Universal Robots URScript: samho_main_Fillet_2023_10_18.script

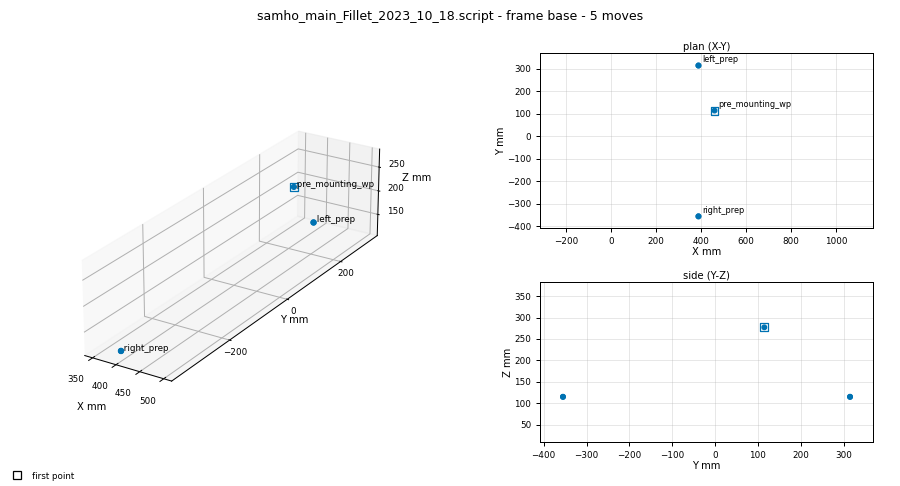
[picture p0: tool path of samho_main_Fillet_2023_10_18.script in frame base, 5 of 121 moves have a stored position in this frame; points joined in program order, loops and branches not executed]
def samho_main_Fillet_2023_10_18():
  set_gravity([0.0, 0.0, 9.82])
  set_standard_analog_input_domain(0, 1)
  set_standard_analog_input_domain(1, 1)
  set_tool_analog_input_domain(0, 1)
  set_tool_analog_input_domain(1, 1)
  set_analog_outputdomain(0, 1)
  set_analog_outputdomain(1, 1)
  set_input_actions_to_default()
  set_tool_digital_input_action(1, "freedrive")
  set_runstate_standard_digital_outputs([0])
  set_runstate_standard_digital_output_to_value(0, 1)
  set_runstate_standard_digital_output_to_value(7, 3)
  step_count_c3da284d_8c38_4948_9d0a_7bbcd1285130 = 0.0
  thread Step_Counter_Thread_b1fbcd7f_a7e8_4366_aae2_1cd96c806efd():
    while (True):
      step_count_c3da284d_8c38_4948_9d0a_7bbcd1285130 = step_count_c3da284d_8c38_4948_9d0a_7bbcd1285130 + 1.0
      sync()
    end
  end
  run Step_Counter_Thread_b1fbcd7f_a7e8_4366_aae2_1cd96c806efd()
  set_safety_mode_transition_hardness(1)
  set_tool_voltage(24)
  set_tcp(p[-0.20748,-9.0E-4,0.38521,1.2569,0.0099,-2.8767])
  set_payload(2.4, [-0.085, 0.00191, 0.125])
  modbus_add_signal("127.0.0.1", 255, 171, 2, "MODBUS_1", False)
  modbus_set_signal_update_frequency("MODBUS_1", 1)
  modbus_add_signal("127.0.0.1", 255, 153, 2, "MODBUS_2", False)
  modbus_set_signal_update_frequency("MODBUS_2", 10)
  modbus_add_signal("127.0.0.1", 255, 154, 2, "MODBUS_3", False)
  modbus_set_signal_update_frequency("MODBUS_3", 10)
  modbus_add_signal("127.0.0.1", 255, 240, 2, "MODBUS_4", False)
  modbus_set_signal_update_frequency("MODBUS_4", 10)
  global A_Touch_trig_l=[False, False, False, False, True, False, False, False, False, False, False]
  global Auto_cur_cell=0
  global last_wv_line=p[0, 0, 0, 0, 0, 0]
  global Auto_trig=False
  global A_Touch_p=[p[0, 0, 0, 0, 0, 0], p[0, 0, 0, 0, 0, 0], p[0, 0, 0, 0, 0, 0], p[0, 0, 0, 0, 0, 0], p[0.52449, -0.29611, -0.03135, -1.44433, -1.03764, -1.44433], p[0, 0, 0, 0, 0, 0], p[0, 0, 0, 0, 0, 0], p[0, 0, 0, 0, 0, 0], p[0, 0, 0, 0, 0, 0], p[0, 0, 0, 0, 0, 0], p[0, 0, 0, 0, 0, 0], p[0, 0, 0, 0, 0, 0], p[0, 0, 0, 0, 0, 0], p[0.5215, -0.2959, 0.14321, -1.44433, -1.03764, -1.44433], p[0, 0, 0, 0, 0, 0], p[0, 0, 0, 0, 0, 0]]
  global last_wv_wp1=p[0, 0, 0, 0, 0, 0]
  global last_pose=p[0, 0, 0, 0, 0, 0]
  global A_Distance_list=[0, 0, 0, 0, 0, 0, 0, 0, 0, 0, 0, 0, 0, 0, 0, 0]
  global Auto_total_cell=1
  global Reset_Trig=False
  global A_Prepos_l=[p[0, 0, 0, 0, 0, 0], p[0, 0, 0, 0, 0, 0], p[0, 0, 0, 0, 0, 0], p[0, 0, 0, 0, 0, 0], p[0.47946, -0.33036, 0.01979, 1.89026, -1.12958, 1.54553], p[0, 0, 0, 0, 0, 0], p[0, 0, 0, 0, 0, 0], p[0, 0, 0, 0, 0, 0], p[0, 0, 0, 0, 0, 0], p[0, 0, 0, 0, 0, 0], p[0, 0, 0, 0, 0, 0], p[0, 0, 0, 0, 0, 0], p[0, 0, 0, 0, 0, 0], p[0, 0, 0, 0, 0, 0], p[0, 0, 0, 0, 0, 0], p[0, 0, 0, 0, 0, 0]]
  global last_z_bottom=0
  global A_Speed_list=[0, 0, 0, 0, 0, 0, 0, 0, 0, 0, 0, 0, 0, 0, 0, 0]
  global Auto_W_num=[4, 0, 0, 0, 0, 0, 0, 0, 0, 0, 0, 0, 0, 0, 0]
  global last_tilt_deg=[0, 0, 0]
  global Base=p[0.0,0.0,0.0,0.0,0.0,0.0]
  global save_timer=0
  global timer_1=0
  def calculate_point_to_move_towards(feature, direction, position_distance):
    local posDir=[direction[0], direction[1], direction[2]]
    if (norm(posDir) < 1e-6):
      return get_target_waypoint()
    end
    local direction_vector_normalized=normalize(posDir)
    local displacement_pose=p[direction_vector_normalized[0] * position_distance,direction_vector_normalized[1] * position_distance,direction_vector_normalized[2] * position_distance,0,0,0]
    local wanted_displacement_in_base_frame=pose_sub(pose_trans(feature, displacement_pose), feature)
    return pose_add(get_target_waypoint(), wanted_displacement_in_base_frame)
  end
  global save_timer_is_counting=False
  global timer_1_is_counting=False
  thread Timer_Thread():
    while (True):
      if (save_timer_is_counting):
        save_timer = save_timer + get_steptime()
      end
      if (timer_1_is_counting):
        timer_1 = timer_1 + get_steptime()
      end
      sync()
    end
  end
  run Timer_Thread()
  def cell_info():
    $ 1483 "cell_info" "noBreak"
    $ 1484 "'cell_setting'"
    # 'cell_setting'
    $ 1485 "a7_f_distance≔get_center"
    global a7_f_distance=get_center
    $ 1486 "'dis + 125'"
    # 'dis + 125'
    $ 1487 "If simulation_mode"
    if (simulation_mode):
      $ 1488 "a6_f_height_l≔190"
      global a6_f_height_l=190
      $ 1489 "a6_f_height_r≔190"
      global a6_f_height_r=190
      $ 1490 "a6_f_width≔690"
      global a6_f_width=690
      $ 1491 "a6_callar_hor≔100"
      global a6_callar_hor=100
      $ 1492 "a6_callar_vert≔100"
      global a6_callar_vert=100
      $ 1493 "center_height≔50"
      global center_height=50
      $ 1494 "EXT_flag1≔integer_to_binary_list(2048)"
      global EXT_flag1= integer_to_binary_list (2048)
      $ 1495 "get_margin_z≔50"
      global get_margin_z=50
    else:
      $ 1496 "Else" "noBreak"
      $ 1497 "a6_f_height_l≔read_port_register(173)"
      global a6_f_height_l= read_port_register (173)
      $ 1498 "a6_f_height_r≔read_port_register(174)"
      global a6_f_height_r= read_port_register (174)
      $ 1499 "a6_f_width≔read_port_register(175)"
      global a6_f_width= read_port_register (175)
      $ 1500 "a6_callar_hor≔read_port_register(181)"
      global a6_callar_hor= read_port_register (181)
      $ 1501 "a6_callar_vert≔read_port_register(182)"
      global a6_callar_vert= read_port_register (182)
      $ 1502 "center_height≔read_port_register(237)"
      global center_height=read_port_register(237)
      $ 1503 "EXT_flag1≔integer_to_binary_list(read_port_register(179))"
      global EXT_flag1= integer_to_binary_list ( read_port_register (179))
      $ 1505 "get_margin_z≔read_port_register(238)"
      global get_margin_z=read_port_register(238)
      $ 1507 "If center_height>32765"
      if (center_height>32765):
        $ 1508 "center_height≔center_height-65535"
        global center_height=center_height-65535
      end
      $ 1509 "If get_margin_z>32765"
      if (get_margin_z>32765):
        $ 1510 "get_margin_z≔get_margin_z-65535"
        global get_margin_z=get_margin_z-65535
      end
    end
    $ 1511 "Initialization"
    $ 1512 "CELL_ROBOT_DIST≔a7_f_distance"
    global CELL_ROBOT_DIST=a7_f_distance
    $ 1513 "CELL_WIDTH≔a6_f_width"
    global CELL_WIDTH=a6_f_width
  end
  def robotand_cell_initalizat():
    $ 1514 "robotand_cell_initalizat" "noBreak"
    $ 1515 "If Auto_trig≟ True "
    if (Auto_trig ==   True  ):
      $ 1516 "Auto_trig≔ False "
      global Auto_trig=  False
      $ 1517 "init"
      $ 1518 "write_port_register(cell_3f_2f_151,0)"
      write_port_register(cell_3f_2f_151,0)
      $ 1519 "write_port_register(cell_info_152,0)"
      write_port_register(cell_info_152,0)
      $ 1520 "write_port_register(weld_req_153,0)"
      write_port_register(weld_req_153,0)
      $ 1521 "write_port_register(touch_cell_155,0)"
      write_port_register(touch_cell_155,0)
      $ 1522 "write_port_register(touch_num_156,0)"
      write_port_register(touch_num_156,0)
      $ 1523 "write_port_register(touch_done_157,0)"
      write_port_register(touch_done_157,0)
      $ 1524 "write_port_register(weld_done_137,0)"
      write_port_register(weld_done_137,0)
      $ 1525 "write_port_register(135,0)"
      write_port_register(135,0)
      $ 1526 "write_port_register(136,0)"
      write_port_register(136,0)
      $ 1527 "write_port_register(165,0)"
      write_port_register(165,0)
      $ 1528 "write_port_register(166,0)"
      write_port_register(166,0)
      $ 1529 "write_port_register(167,0)"
      write_port_register(167,0)
      $ 1530 "write_port_register(169,0)"
      write_port_register(169,0)
      $ 1531 "write_port_register(170,0)"
      write_port_register(170,0)
      $ 1532 "write_port_register(221,0)"
      write_port_register(221,0)
      $ 1533 "write_port_register(222,0)"
      write_port_register(222,0)
      $ 1534 "write_port_register(223,0)"
      write_port_register(223,0)
      $ 1535 "write_port_register(224,0)"
      write_port_register(224,0)
      $ 1536 "write_port_register(225,0)"
      write_port_register(225,0)
      $ 1537 "write_port_register(226,0)"
      write_port_register(226,0)
      $ 1538 "write_port_register(227,0)"
      write_port_register(227,0)
      $ 1539 "write_port_register(228,0)"
      write_port_register(228,0)
      $ 1540 "write_port_register(240,0)"
      write_port_register(240,0)
      $ 1541 "write_port_register(176,0)"
      write_port_register(176,0)
      $ 1542 "write_port_register(177,0)"
      write_port_register(177,0)
      $ 1543 "write_port_register(154,0)"
      write_port_register(154,0)
    end
    $ 1544 "sync()"
    sync()
  end
  def welding_parameter_init():
    $ 1545 "welding_parameter_init" "noBreak"
    $ 1546 "init"
    $ 1547 "If A_sel_v≟A_VL1 or A_sel_v≟A_VL2 or A_sel_v≟A_VR1 or A_sel_v≟A_VR2"
    if (A_sel_v == A_VL1  or  A_sel_v == A_VL2  or  A_sel_v == A_VR1  or  A_sel_v == A_VR2):
      $ 1548 "position_3f2f≔position_3F"
      global position_3f2f=position_3F
      $ 1549 "write_port_register(cell_3f_2f_151,A_sel_v)"
      write_port_register(cell_3f_2f_151,A_sel_v)
      $ 1550 "b8_wv_2f≔ False "
      global b8_wv_2f=  False
      $ 1551 "d_lean_degree≔0"
      global d_lean_degree=0
    else:
      $ 1552 "Else" "noBreak"
      $ 1553 "position_3f2f≔position_2F"
      global position_3f2f=position_2F
      $ 1554 "b8_wv_2f≔ True "
      global b8_wv_2f=  True
      $ 1555 "d_lean_degree≔30"
      global d_lean_degree=30
      $ 1556 "write_port_register(cell_3f_2f_151,A_HOR)"
      write_port_register(cell_3f_2f_151,A_HOR)
    end
    $ 1557 "If current_path≥2"
    if (current_path >= 2):
      $ 1558 "write_port_register(cell_info_152,current_path)"
      write_port_register(cell_info_152,current_path)
    else:
      $ 1559 "Else" "noBreak"
      $ 1560 "write_port_register(cell_info_152,1)"
      write_port_register(cell_info_152,1)
    end
    $ 1561 "write_port_register(return_done_240,0)"
    write_port_register(return_done_240,0)
    $ 1562 "Wait: 0.3"
    sleep(0.3)
    $ 1563 "write_port_register(weld_req_153,1)"
    write_port_register(weld_req_153,1)
    $ 1564 "Wait read_port_register(return_done_240)≟1"
    while (not( read_port_register (return_done_240) == 1)):
      sync()
    end
    $ 1565 "write_port_register(weld_req_153,0)"
    write_port_register(weld_req_153,0)
    $ 1566 "touch_m_check≔0"
    global touch_m_check=0
    $ 1567 "start_end_from_pendant"
    $ 1568 "d_start_current≔read_port_register(244)/10"
    global d_start_current= read_port_register (244)/10
    $ 1569 "d_start_voltage≔read_port_register(245)/10"
    global d_start_voltage= read_port_register (245)/10
    $ 1570 "d_start_time≔read_port_register(241)/10"
    global d_start_time= read_port_register (241)/10
    $ 1571 "d_end_current≔read_port_register(249)/10"
    global d_end_current= read_port_register (249)/10
    $ 1572 "d_end_voltage≔read_port_register(250)/10"
    global d_end_voltage= read_port_register (250)/10
    $ 1573 "d_end_time≔read_port_register(246)/10"
    global d_end_time= read_port_register (246)/10
    $ 1574 "d_end_current_2≔read_port_register(254)/10"
    global d_end_current_2= read_port_register (254)/10
    $ 1575 "d_end_voltage_2≔read_port_register(255)/10"
    global d_end_voltage_2= read_port_register (255)/10
    $ 1576 "d_end_time_2≔read_port_register(251)/10"
    global d_end_time_2= read_port_register (251)/10
    $ 1577 "a7_weld_crater≔[d_start_current,d_start_voltage,d_start_time,d_end_current,d_end_voltage,d_end_time,d_lean_degree]"
    global a7_weld_crater=[d_start_current,d_start_voltage,d_start_time,d_end_current,d_end_voltage,d_end_time,d_lean_degree]
    $ 1578 "a0_volt_ref≔read_port_register(231)/10"
    global a0_volt_ref= read_port_register (231)/10
    $ 1579 "a1_amp_ref≔read_port_register(232)/10"
    global a1_amp_ref= read_port_register (232)/10
    $ 1580 "a2_speed_cpm≔read_port_register(233)/10"
    global a2_speed_cpm= read_port_register (233)/10
    $ 1581 "a3_wv_amplitude≔read_port_register(234)/10"
    global a3_wv_amplitude= read_port_register (234)/10
    $ 1582 "a4_wv_frequency≔read_port_register(225)/10"
    global a4_wv_frequency= read_port_register (225)/10
    $ 1583 "b1_appro_param≔0"
    global b1_appro_param=0
    $ 1584 "b4_wv_delay2≔read_port_register(226)/10"
    global b4_wv_delay2= read_port_register (226)/10
    $ 1585 "b6_wv_delay4≔read_port_register(227)/10"
    global b6_wv_delay4= read_port_register (227)/10
    $ 1586 "b3_wv_delay1≔0"
    global b3_wv_delay1=0
    $ 1587 "b5_wv_delay3≔0"
    global b5_wv_delay3=0
    $ 1588 "b3_dealy_all≔[b3_wv_delay1,b4_wv_delay2,b5_wv_delay3,b6_wv_delay4]"
    global b3_dealy_all=[b3_wv_delay1,b4_wv_delay2,b5_wv_delay3,b6_wv_delay4]
    $ 1589 "get_width_182≔read_port_register(182)"
    global get_width_182= read_port_register (182)
    $ 1590 "b9_touch_sens≔20"
    global b9_touch_sens=20
    $ 1591 "task_angle≔register_read(228)/10"
    global task_angle=register_read(228)/10
    $ 1592 "Circle_Speed≔a2_speed_cpm"
    global Circle_Speed=a2_speed_cpm
    $ 1593 "CELL_BOTTOM≔a7_cell_bottom"
    global CELL_BOTTOM=a7_cell_bottom
    $ 1594 "a6_scallup_left≔read_port_register(176)"
    global a6_scallup_left= read_port_register (176)
    $ 1595 "a6_scallup_righ≔read_port_register(177)"
    global a6_scallup_righ= read_port_register (177)
    $ 1596 "a5_f_hole≔[a7_cell_bottom,a6_scallup_left,a6_scallup_righ]"
    global a5_f_hole=[a7_cell_bottom,a6_scallup_left,a6_scallup_righ]
    $ 1630 "폴더"
    $ 1631 "offset_2f_x≔7"
    global offset_2f_x=7
    $ 1632 "offset_3f_z≔-5"
    global offset_3f_z=-5
    $ 1633 "If A_sel_v≟A_VR1 or A_sel_v≟A_VR2"
    if (A_sel_v == A_VR1  or  A_sel_v == A_VR2):
      $ 1634 "'3F'"
      # '3F'
      $ 1635 "b2_left_par≔ False "
      global b2_left_par=  False
      $ 1636 "b8_wv_type≔1"
      global b8_wv_type=1
      $ 1637 "If A_sel_v≟A_VR2 and (b1_cell_info_R≟c or b1_cell_info_R≟d)"
      if (A_sel_v == A_VR2  and  (b1_cell_info_R == c  or  b1_cell_info_R == d)):
        $ 1638 "b7_tilt_degree≔[0,0,0]"
        global b7_tilt_degree=[0,0,0]
      else:
        $ 1639 "Else" "noBreak"
        $ 1640 "b7_tilt_degree≔[task_angle,-27,0]"
        global b7_tilt_degree=[task_angle,-27,0]
      end
      $ 1641 "c3_arc_enable≔1"
      global c3_arc_enable=1
    else:
      $ 1642 "ElseIf A_sel_v≟A_VL1 or A_sel_v≟A_VL2"
      if (A_sel_v == A_VL1  or  A_sel_v == A_VL2):
        $ 1643 "'3F'"
        # '3F'
        $ 1644 "b2_left_par≔ True "
        global b2_left_par=  True
        $ 1645 "b8_wv_type≔1"
        global b8_wv_type=1
        $ 1646 "If A_sel_v≟A_VL2 and (b1_cell_info_L≟c or b1_cell_info_L≟d)"
        if (A_sel_v == A_VL2  and  (b1_cell_info_L == c  or  b1_cell_info_L == d)):
          $ 1647 "b7_tilt_degree≔[0,0,0]"
          global b7_tilt_degree=[0,0,0]
        else:
          $ 1648 "Else" "noBreak"
          $ 1649 "b7_tilt_degree≔[task_angle,-27,0]"
          global b7_tilt_degree=[task_angle,-27,0]
        end
        $ 1650 "c3_arc_enable≔1"
        global c3_arc_enable=1
      else:
        $ 1651 "Else" "noBreak"
        $ 1652 "b2_left_par≔ True "
        global b2_left_par=  True
        $ 1653 "b8_wv_type≔2"
        global b8_wv_type=2
        $ 1654 "If A_sel_v≟A_HOR"
        if (A_sel_v == A_HOR):
          $ 1655 "b7_tilt_degree≔[30,-1*task_angle,0]"
          global b7_tilt_degree=[30,-1*task_angle,0]
        else:
          $ 1656 "Else" "noBreak"
          $ 1658 "b7_tilt_degree≔[30,-1*task_angle,0]"
          global b7_tilt_degree=[30,-1*task_angle,0]
        end
        $ 1660 "c3_arc_enable≔0"
        global c3_arc_enable=0
      end
    end
    $ 1661 "If A_sel_v≟A_VL2 or A_sel_v≟A_VR2"
    if (A_sel_v == A_VL2  or  A_sel_v == A_VR2):
      $ 1662 "If b1_cell_info_L≟E or b1_cell_info_L≟e or b1_cell_info_R≟E or b1_cell_info_R≟e"
      if (b1_cell_info_L == E  or  b1_cell_info_L == e  or  b1_cell_info_R == E  or  b1_cell_info_R == e):
        $ 1663 "a8_wv_distance≔read_port_register(182)-a5_f_hole[1]-offset_3f_begin"
        global a8_wv_distance= read_port_register (182)-a5_f_hole[1]-offset_3f_begin
      else:
        $ 1664 "Else" "noBreak"
        $ 1665 "a8_wv_distance≔read_port_register(182)-offset_3f_begin"
        global a8_wv_distance= read_port_register (182)-offset_3f_begin
      end
    else:
      $ 1670 "Else" "noBreak"
      $ 1671 "If b2_left_par"
      if (b2_left_par):
        $ 1672 "Comment"
        # Comment
        $ 1673 "a8_wv_distance≔a6_f_height_l-a5_f_hole[1]-offset_3f_begin"
        global a8_wv_distance=a6_f_height_l-a5_f_hole[1]-offset_3f_begin
        $ 1674 "Comment"
        # Comment
      else:
        $ 1675 "Else" "noBreak"
        $ 1676 "a8_wv_distance≔a6_f_height_r-a5_f_hole[1]-offset_3f_begin"
        global a8_wv_distance=a6_f_height_r-a5_f_hole[1]-offset_3f_begin
      end
    end
    $ 1677 "Ext fun & Squash"
    $ 1678 "If (A_sel_v≟A_VL1 or A_sel_v≟A_VL2) and (b1_cell_info_L≟B or b1_cell_info_L≟D)"
    if ((A_sel_v == A_VL1  or  A_sel_v == A_VL2)  and  (b1_cell_info_L == B  or  b1_cell_info_L == D)):
      $ 1679 "Scallup_check≔ True "
      global Scallup_check=  True
    else:
      $ 1680 "ElseIf (A_sel_v≟A_VR1 or A_sel_v≟A_VR2) and (b1_cell_info_R≟B or b1_cell_info_R≟D)"
      if ((A_sel_v == A_VR1  or  A_sel_v == A_VR2)  and  (b1_cell_info_R == B  or  b1_cell_info_R == D)):
        $ 1681 "Scallup_check≔ True "
        global Scallup_check=  True
      else:
        $ 1682 "Else" "noBreak"
        $ 1683 "Scallup_check≔ False "
        global Scallup_check=  False
      end
    end
    $ 1684 "If (EXT_flag1[7]≟ True ) and (A_sel_v≠A_HOR) and (A_sel_v≠A_VL2) and (A_sel_v≠A_VR2) and (Scallup_check≟ False )"
    if ((EXT_flag1[7] ==   True  )  and  (A_sel_v != A_HOR)  and  (A_sel_v != A_VL2)  and  (A_sel_v != A_VR2)  and  (Scallup_check ==   False  )):
      $ 1685 "squash"
      $ 1686 "squash_enable≔1"
      global squash_enable=1
      $ 1687 "squash_voltage≔24.5"
      global squash_voltage=24.5
      $ 1688 "squash_current≔190"
      global squash_current=190
      $ 1689 "squash_amp≔7"
      global squash_amp=7
      $ 1690 "squash_speed≔10"
      global squash_speed=10
      $ 1691 "squash_cycle≔8"
      global squash_cycle=8
    else:
      $ 1692 "Else" "noBreak"
      $ 1693 "squash"
      $ 1694 "squash_enable≔0"
      global squash_enable=0
      $ 1695 "squash_voltage≔0"
      global squash_voltage=0
      $ 1696 "squash_current≔0"
      global squash_current=0
      $ 1697 "squash_amp≔0"
      global squash_amp=0
      $ 1698 "squash_speed≔0"
      global squash_speed=0
      $ 1699 "squash_cycle≔0"
      global squash_cycle=0
    end
    $ 1700 "If EXT_flag1[8]≟ True  and EXT_flag1[9]≟ False "
    if (EXT_flag1[8] ==   True    and  EXT_flag1[9] ==   False  ):
      $ 1701 "sludge≔1"
      global sludge=1
    else:
      $ 1702 "ElseIf EXT_flag1[8]≟ False  and EXT_flag1[9]≟ True "
      if (EXT_flag1[8] ==   False    and  EXT_flag1[9] ==   True  ):
        $ 1703 "sludge≔2"
        global sludge=2
      else:
        $ 1704 "Else" "noBreak"
        $ 1705 "sludge≔0"
        global sludge=0
      end
    end
    $ 1706 "waste_cycle≔2"
    global waste_cycle=2
    $ 1707 "c0_offset_x≔read_port_register(229)/10"
    global c0_offset_x= read_port_register (229)/10
    $ 1708 "c0_offset_z≔read_port_register(230)/10"
    global c0_offset_z= read_port_register (230)/10
    $ 1709 "squash_l≔[a0_volt_ref,a1_amp_ref,squash_enable,squash_voltage,squash_current,squash_amp,squash_speed,squash_cycle,waste_cycle,c0_offset_x,c0_offset_z]"
    global squash_l=[a0_volt_ref,a1_amp_ref,squash_enable,squash_voltage,squash_current,squash_amp,squash_speed,squash_cycle,waste_cycle,c0_offset_x,c0_offset_z]
    $ 1710 "WV_gap"
    $ 1711 "c5_wv_gap_y≔read_port_register(236)/10"
    global c5_wv_gap_y= read_port_register (236)/10
    $ 1712 "c6_wv_gap_cpm≔read_port_register(235)/10"
    global c6_wv_gap_cpm= read_port_register (235)/10
    $ 1713 "c9_wv_gap_freq≔a4_wv_frequency"
    global c9_wv_gap_freq=a4_wv_frequency
    $ 1714 "If c6_wv_gap_cpm≟a2_speed_cpm and a3_wv_amplitude≟c5_wv_gap_y"
    if (c6_wv_gap_cpm == a2_speed_cpm  and  a3_wv_amplitude == c5_wv_gap_y):
      $ 1715 "c4_gap_enable≔0"
      global c4_gap_enable=0
    else:
      $ 1716 "Else" "noBreak"
      $ 1717 "c4_gap_enable≔1"
      global c4_gap_enable=1
    end
    $ 1718 "c7_wv_gap≔[c4_gap_enable,c5_wv_gap_y,c6_wv_gap_cpm,c9_wv_gap_freq]"
    global c7_wv_gap=[c4_gap_enable,c5_wv_gap_y,c6_wv_gap_cpm,c9_wv_gap_freq]
    $ 1719 "arc_sen"
    $ 1720 "c3_X_p_gain≔read_port_register(186)/10"
    global c3_X_p_gain= read_port_register (186)/10
    $ 1721 "c3_X_i_gain≔read_port_register(187)/10"
    global c3_X_i_gain= read_port_register (187)/10
    $ 1722 "c3_Z_p_gain≔read_port_register(184)/10"
    global c3_Z_p_gain= read_port_register (184)/10
    $ 1723 "c3_Z_i_gain≔read_port_register(185)/10"
    global c3_Z_i_gain= read_port_register (185)/10
    $ 1724 "c3_wv_arc_fix≔0"
    global c3_wv_arc_fix=0
    $ 1725 "c3_wv_arc≔[c3_arc_enable,c3_X_p_gain,c3_X_i_gain,c3_Z_p_gain,c3_Z_i_gain,c3_wv_arc_fix]"
    global c3_wv_arc=[c3_arc_enable,c3_X_p_gain,c3_X_i_gain,c3_Z_p_gain,c3_Z_i_gain,c3_wv_arc_fix]
    $ 1726 "volt and current"
    $ 1727 "set_current_voltage(a1_amp_ref,a0_volt_ref)"
    set_current_voltage(a1_amp_ref,a0_volt_ref)
    $ 1728 "write_port_register(154,1)"
    write_port_register(154,1)
    $ 1729 "Wait read_port_register(return_done_240)≟0"
    while (not( read_port_register (return_done_240) == 0)):
      sync()
    end
    $ 1730 "write_port_register(154,0)"
    write_port_register(154,0)
  end
  def welding_parameter_sim():
    $ 1731 "welding_parameter_sim" "noBreak"
    $ 1732 "init"
    $ 1733 "If A_sel_v≟A_VL1 or A_sel_v≟A_VL2 or A_sel_v≟A_VR1 or A_sel_v≟A_VR2"
    if (A_sel_v == A_VL1  or  A_sel_v == A_VL2  or  A_sel_v == A_VR1  or  A_sel_v == A_VR2):
      $ 1734 "position_3f2f≔position_3F"
      global position_3f2f=position_3F
      $ 1735 "write_port_register(cell_3f_2f_151,A_sel_v)"
      write_port_register(cell_3f_2f_151,A_sel_v)
      $ 1736 "b8_wv_2f≔ False "
      global b8_wv_2f=  False
      $ 1737 "d_lean_degree≔0"
      global d_lean_degree=0
    else:
      $ 1738 "Else" "noBreak"
      $ 1739 "position_3f2f≔position_2F"
      global position_3f2f=position_2F
      $ 1740 "b8_wv_2f≔ True "
      global b8_wv_2f=  True
      $ 1741 "d_lean_degree≔30"
      global d_lean_degree=30
      $ 1742 "write_port_register(cell_3f_2f_151,A_HOR)"
      write_port_register(cell_3f_2f_151,A_HOR)
    end
    $ 1743 "If current_path≥2"
    if (current_path >= 2):
      $ 1744 "write_port_register(cell_info_152,current_path)"
      write_port_register(cell_info_152,current_path)
    else:
      $ 1745 "Else" "noBreak"
      $ 1746 "write_port_register(cell_info_152,1)"
      write_port_register(cell_info_152,1)
    end
    $ 1747 "write_port_register(return_done_240,0)"
    write_port_register(return_done_240,0)
    $ 1748 "Wait: 0.3"
    sleep(0.3)
    $ 1749 "write_port_register(weld_req_153,1)"
    write_port_register(weld_req_153,1)
    $ 1751 "write_port_register(weld_req_153,0)"
    write_port_register(weld_req_153,0)
    $ 1752 "touch_m_check≔0"
    global touch_m_check=0
    $ 1753 "start_end_from_pendant"
    $ 1754 "d_start_current≔read_port_register(244)/10"
    global d_start_current= read_port_register (244)/10
    $ 1755 "d_start_voltage≔read_port_register(245)/10"
    global d_start_voltage= read_port_register (245)/10
    $ 1756 "d_start_time≔read_port_register(241)/10"
    global d_start_time= read_port_register (241)/10
    $ 1757 "d_end_current≔read_port_register(249)/10"
    global d_end_current= read_port_register (249)/10
    $ 1758 "d_end_voltage≔read_port_register(250)/10"
    global d_end_voltage= read_port_register (250)/10
    $ 1759 "d_end_time≔read_port_register(246)/10"
    global d_end_time= read_port_register (246)/10
    $ 1760 "d_end_current_2≔read_port_register(254)/10"
    global d_end_current_2= read_port_register (254)/10
    $ 1761 "d_end_voltage_2≔read_port_register(255)/10"
    global d_end_voltage_2= read_port_register (255)/10
    $ 1762 "d_end_time_2≔read_port_register(251)/10"
    global d_end_time_2= read_port_register (251)/10
    $ 1763 "a7_weld_crater≔[d_start_current,d_start_voltage,d_start_time,d_end_current,d_end_voltage,d_end_time,d_lean_degree]"
    global a7_weld_crater=[d_start_current,d_start_voltage,d_start_time,d_end_current,d_end_voltage,d_end_time,d_lean_degree]
    $ 1764 "a0_volt_ref≔read_port_register(231)/10"
    global a0_volt_ref= read_port_register (231)/10
    $ 1765 "a1_amp_ref≔read_port_register(232)/10"
    global a1_amp_ref= read_port_register (232)/10
    $ 1766 "b1_appro_param≔0"
    global b1_appro_param=0
    $ 1767 "Folder"
    $ 1768 "a2_speed_cpm≔17"
    global a2_speed_cpm=17
    $ 1769 "a3_wv_amplitude≔5"
    global a3_wv_amplitude=5
    $ 1770 "a4_wv_frequency≔1.4"
    global a4_wv_frequency=1.4
    $ 1771 "b4_wv_delay2≔0.3"
    global b4_wv_delay2=0.3
    $ 1772 "b6_wv_delay4≔0.3"
    global b6_wv_delay4=0.3
    $ 1773 "b9_touch_sens≔10"
    global b9_touch_sens=10
    $ 1774 "task_angle≔0"
    global task_angle=0
    $ 1775 "a6_scallup_left≔0"
    global a6_scallup_left=0
    $ 1776 "a6_scallup_righ≔0"
    global a6_scallup_righ=0
    $ 1777 "b3_wv_delay1≔0"
    global b3_wv_delay1=0
    $ 1778 "b5_wv_delay3≔0"
    global b5_wv_delay3=0
    $ 1779 "b3_dealy_all≔[b3_wv_delay1,b4_wv_delay2,b5_wv_delay3,b6_wv_delay4]"
    global b3_dealy_all=[b3_wv_delay1,b4_wv_delay2,b5_wv_delay3,b6_wv_delay4]
    $ 1780 "get_width_182≔a6_callar_vert"
    global get_width_182=a6_callar_vert
    $ 1781 "task_angle≔register_read(228)/10"
    global task_angle=register_read(228)/10
    $ 1782 "Circle_Speed≔a2_speed_cpm"
    global Circle_Speed=a2_speed_cpm
    $ 1783 "CELL_BOTTOM≔a7_cell_bottom"
    global CELL_BOTTOM=a7_cell_bottom
    $ 1784 "a5_f_hole≔[a7_cell_bottom,a6_scallup_left,a6_scallup_righ]"
    global a5_f_hole=[a7_cell_bottom,a6_scallup_left,a6_scallup_righ]
    $ 1785 "폴더"
    $ 1786 "offset_2f_x≔7"
    global offset_2f_x=7
    $ 1787 "offset_3f_z≔-5"
    global offset_3f_z=-5
    $ 1788 "If A_sel_v≟A_VR1 or A_sel_v≟A_VR2"
    if (A_sel_v == A_VR1  or  A_sel_v == A_VR2):
      $ 1789 "'3F'"
      # '3F'
      $ 1790 "b2_left_par≔ False "
      global b2_left_par=  False
      $ 1791 "b8_wv_type≔1"
      global b8_wv_type=1
      $ 1792 "b7_tilt_degree≔[task_angle,-27,0]"
      global b7_tilt_degree=[task_angle,-27,0]
      $ 1793 "c3_arc_enable≔1"
      global c3_arc_enable=1
    else:
      $ 1794 "ElseIf A_sel_v≟A_VL1 or A_sel_v≟A_VL2"
      if (A_sel_v == A_VL1  or  A_sel_v == A_VL2):
        $ 1795 "'3F'"
        # '3F'
        $ 1796 "b2_left_par≔ True "
        global b2_left_par=  True
        $ 1797 "b8_wv_type≔1"
        global b8_wv_type=1
        $ 1798 "b7_tilt_degree≔[task_angle,-27,0]"
        global b7_tilt_degree=[task_angle,-27,0]
        $ 1799 "c3_arc_enable≔1"
        global c3_arc_enable=1
      else:
        $ 1800 "Else" "noBreak"
        $ 1801 "b2_left_par≔ True "
        global b2_left_par=  True
        $ 1802 "b8_wv_type≔2"
        global b8_wv_type=2
        $ 1803 "b7_tilt_degree≔[30,-1*task_angle,0]"
        global b7_tilt_degree=[30,-1*task_angle,0]
        $ 1805 "c3_arc_enable≔0"
        global c3_arc_enable=0
      end
    end
    $ 1806 "If A_sel_v≟A_VL2 or A_sel_v≟A_VR2"
    if (A_sel_v == A_VL2  or  A_sel_v == A_VR2):
      $ 1807 "a8_wv_distance≔read_port_register(182)"
      global a8_wv_distance= read_port_register (182)
    else:
      $ 1812 "Else" "noBreak"
      $ 1813 "If b2_left_par"
      if (b2_left_par):
        $ 1814 "Comment"
        # Comment
        $ 1815 "a8_wv_distance≔a6_f_height_l-a5_f_hole[1]"
        global a8_wv_distance=a6_f_height_l-a5_f_hole[1]
        $ 1816 "Comment"
        # Comment
      else:
        $ 1817 "Else" "noBreak"
        $ 1818 "a8_wv_distance≔a6_f_height_r-a5_f_hole[1]"
        global a8_wv_distance=a6_f_height_r-a5_f_hole[1]
      end
    end
    $ 1819 "Ext fun & Squash"
    $ 1820 "If (A_sel_v≟A_VL1 or A_sel_v≟A_VL2) and (b1_cell_info_L≟B or b1_cell_info_L≟D)"
    if ((A_sel_v == A_VL1  or  A_sel_v == A_VL2)  and  (b1_cell_info_L == B  or  b1_cell_info_L == D)):
      $ 1821 "Scallup_check≔ True "
      global Scallup_check=  True
    else:
      $ 1822 "ElseIf (A_sel_v≟A_VR1 or A_sel_v≟A_VR2) and (b1_cell_info_R≟B or b1_cell_info_R≟D)"
      if ((A_sel_v == A_VR1  or  A_sel_v == A_VR2)  and  (b1_cell_info_R == B  or  b1_cell_info_R == D)):
        $ 1823 "Scallup_check≔ True "
        global Scallup_check=  True
      else:
        $ 1824 "Else" "noBreak"
        $ 1825 "Scallup_check≔ False "
        global Scallup_check=  False
      end
    end
    $ 1826 "If (EXT_flag1[7]≟ True ) and (A_sel_v≠A_HOR) and (A_sel_v≠A_VL2) and (A_sel_v≠A_VR2) and (Scallup_check≟ False )"
    if ((EXT_flag1[7] ==   True  )  and  (A_sel_v != A_HOR)  and  (A_sel_v != A_VL2)  and  (A_sel_v != A_VR2)  and  (Scallup_check ==   False  )):
      $ 1827 "squash"
      $ 1828 "squash_enable≔1"
      global squash_enable=1
      $ 1829 "squash_voltage≔24.5"
      global squash_voltage=24.5
      $ 1830 "squash_current≔190"
      global squash_current=190
      $ 1831 "squash_amp≔7"
      global squash_amp=7
      $ 1832 "squash_speed≔10"
      global squash_speed=10
      $ 1833 "squash_cycle≔8"
      global squash_cycle=8
    else:
      $ 1834 "Else" "noBreak"
      $ 1835 "squash"
      $ 1836 "squash_enable≔0"
      global squash_enable=0
      $ 1837 "squash_voltage≔0"
      global squash_voltage=0
      $ 1838 "squash_current≔0"
      global squash_current=0
      $ 1839 "squash_amp≔0"
      global squash_amp=0
      $ 1840 "squash_speed≔0"
      global squash_speed=0
      $ 1841 "squash_cycle≔0"
      global squash_cycle=0
    end
    $ 1842 "waste_cycle≔2"
    global waste_cycle=2
    $ 1843 "c0_offset_x≔read_port_register(229)/10"
    global c0_offset_x= read_port_register (229)/10
    $ 1844 "c0_offset_z≔read_port_register(230)/10"
    global c0_offset_z= read_port_register (230)/10
    $ 1845 "squash_l≔[a0_volt_ref,a1_amp_ref,squash_enable,squash_voltage,squash_current,squash_amp,squash_speed,squash_cycle,waste_cycle,c0_offset_x,c0_offset_z]"
    global squash_l=[a0_volt_ref,a1_amp_ref,squash_enable,squash_voltage,squash_current,squash_amp,squash_speed,squash_cycle,waste_cycle,c0_offset_x,c0_offset_z]
    $ 1846 "WV_gap"
    $ 1847 "c5_wv_gap_y≔a3_wv_amplitude"
    global c5_wv_gap_y=a3_wv_amplitude
    $ 1848 "c6_wv_gap_cpm≔a2_speed_cpm"
    global c6_wv_gap_cpm=a2_speed_cpm
    $ 1849 "c9_wv_gap_freq≔a4_wv_frequency"
    global c9_wv_gap_freq=a4_wv_frequency
    $ 1850 "If c6_wv_gap_cpm≟a2_speed_cpm and a3_wv_amplitude≟c5_wv_gap_y"
    if (c6_wv_gap_cpm == a2_speed_cpm  and  a3_wv_amplitude == c5_wv_gap_y):
      $ 1851 "c4_gap_enable≔0"
      global c4_gap_enable=0
    else:
      $ 1852 "Else" "noBreak"
      $ 1853 "c4_gap_enable≔1"
      global c4_gap_enable=1
    end
    $ 1854 "c4_gap_enable≔0"
    global c4_gap_enable=0
    $ 1855 "c7_wv_gap≔[c4_gap_enable,c5_wv_gap_y,c6_wv_gap_cpm,c9_wv_gap_freq]"
    global c7_wv_gap=[c4_gap_enable,c5_wv_gap_y,c6_wv_gap_cpm,c9_wv_gap_freq]
    $ 1856 "arc_sen"
    $ 1857 "c3_X_p_gain≔read_port_register(186)/10"
    global c3_X_p_gain= read_port_register (186)/10
    $ 1858 "c3_X_i_gain≔read_port_register(187)/10"
    global c3_X_i_gain= read_port_register (187)/10
    $ 1859 "c3_Z_p_gain≔read_port_register(184)/10"
    global c3_Z_p_gain= read_port_register (184)/10
    $ 1860 "c3_Z_i_gain≔read_port_register(185)/10"
    global c3_Z_i_gain= read_port_register (185)/10
    $ 1861 "c3_wv_arc_fix≔0"
    global c3_wv_arc_fix=0
    $ 1862 "c3_wv_arc≔[c3_arc_enable,c3_X_p_gain,c3_X_i_gain,c3_Z_p_gain,c3_Z_i_gain,c3_wv_arc_fix]"
    global c3_wv_arc=[c3_arc_enable,c3_X_p_gain,c3_X_i_gain,c3_Z_p_gain,c3_Z_i_gain,c3_wv_arc_fix]
    $ 1863 "volt and current"
    $ 1864 "set_current_voltage(a1_amp_ref,a0_volt_ref)"
    set_current_voltage(a1_amp_ref,a0_volt_ref)
    $ 1865 "write_port_register(154,1)"
    write_port_register(154,1)
    $ 1867 "write_port_register(154,0)"
    write_port_register(154,0)
  end
  def Move_done():
    $ 1868 "Move_done" "noBreak"
    $ 1869 "write_port_register(robot_move_163,0)"
    write_port_register(robot_move_163,0)
    $ 1870 "write_port_register(robot_pose_164,0)"
    write_port_register(robot_pose_164,0)
    $ 1871 "write_port_register(robot_ready_141,1)"
    write_port_register(robot_ready_141,1)
  end
  def MoveFun():
    $ 1872 "MoveFun" "noBreak"
    $ 1873 "b_touch_pos≔A_Prepos_l[A_sel_v]"
    global b_touch_pos=A_Prepos_l[A_sel_v]
    $ 1874 "MoveL"
    $ 1875 "b_touch_pos" "breakAfter"
    movel(pose_trans(Base, b_touch_pos), a=0.35, v=0.35)
  end
  def MoveFun_cd():
    $ 1876 "MoveFun_cd" "noBreak"
    $ 1877 "b_touch_pos≔A_Prepos_l[A_sel_v]"
    global b_touch_pos=A_Prepos_l[A_sel_v]
    $ 1878 "If A_sel_v≟A_VR2 and (b1_cell_info_R≟c or b1_cell_info_R≟d)"
    if (A_sel_v == A_VR2  and  (b1_cell_info_R == c  or  b1_cell_info_R == d)):
      $ 1879 "tilt_deg≔27"
      global tilt_deg=27
      $ 1880 "tilt_deg_ry≔19"
      global tilt_deg_ry=19
      $ 1881 "tilt_deg_rz≔0"
      global tilt_deg_rz=0
    else:
      $ 1882 "Else" "noBreak"
      $ 1883 "tilt_deg≔10"
      global tilt_deg=10
      $ 1884 "tilt_deg_ry≔5"
      global tilt_deg_ry=5
      $ 1885 "tilt_deg_rz≔0"
      global tilt_deg_rz=0
    end
    $ 1886 "If b2_left_par"
    if (b2_left_par):
      $ 1887 "b_touch_pos≔pose_add(b_touch_pos, p[0,18/1000,0,0,0,0])"
      global b_touch_pos= pose_add (b_touch_pos, p[0,18/1000,0,0,0,0])
      $ 1888 "b_touch_pos≔pose_trans(b_touch_pos, p[0,0,0,d2r(-tilt_deg),d2r(-tilt_deg_ry),d2r(tilt_deg_rz)])"
      global b_touch_pos= pose_trans (b_touch_pos, p[0,0,0,d2r(-tilt_deg),d2r(-tilt_deg_ry),d2r(tilt_deg_rz)])
    else:
      $ 1889 "Else" "noBreak"
      $ 1890 "b_touch_pos≔pose_add(b_touch_pos, p[0,-18/1000,0,0,0,0])"
      global b_touch_pos= pose_add (b_touch_pos, p[0,-18/1000,0,0,0,0])
      $ 1891 "b_touch_pos≔pose_trans(b_touch_pos, p[0,0,0,d2r(tilt_deg),d2r(-tilt_deg_ry),d2r(-tilt_deg_rz)])"
      global b_touch_pos= pose_trans (b_touch_pos, p[0,0,0,d2r(tilt_deg),d2r(-tilt_deg_ry),d2r(-tilt_deg_rz)])
    end
    $ 1892 "MoveL"
    $ 1893 "b_touch_pos" "breakAfter"
    movel(pose_trans(Base, b_touch_pos), a=0.35, v=0.35)
  end
  def MoveandTouchFun_2f():
    $ 1894 "MoveandTouchFun_2f" "noBreak"
    $ 1895 "b_touch_pos≔A_Prepos_l[A_sel_v]"
    global b_touch_pos=A_Prepos_l[A_sel_v]
    $ 1896 "tilt_deg≔3"
    global tilt_deg=3
    $ 1897 "tilt_deg_ry≔3"
    global tilt_deg_ry=3
    $ 1898 "tilt_deg_rz≔0"
    global tilt_deg_rz=0
    $ 1899 "If b2_left_par"
    if (b2_left_par):
      $ 1900 "b_touch_pos≔pose_trans(b_touch_pos, p[0,0/1000,0,d2r(tilt_deg),d2r(-tilt_deg_ry),d2r(tilt_deg_rz)])"
      global b_touch_pos= pose_trans (b_touch_pos, p[0,0/1000,0,d2r(tilt_deg),d2r(-tilt_deg_ry),d2r(tilt_deg_rz)])
    else:
      $ 1901 "Else" "noBreak"
      $ 1902 "b_touch_pos≔pose_trans(b_touch_pos, p[0,0/1000,0,d2r(tilt_deg),d2r(-tilt_deg_ry),d2r(-tilt_deg_rz)])"
      global b_touch_pos= pose_trans (b_touch_pos, p[0,0/1000,0,d2r(tilt_deg),d2r(-tilt_deg_ry),d2r(-tilt_deg_rz)])
    end
    $ 1903 "MoveL"
    $ 1904 "b_touch_pos" "breakAfter"
    movel(pose_trans(Base, b_touch_pos), a=0.35, v=0.35)
    $ 1905 "Touch_2f"
    $ 1906 "touch_result≔touch_fun_2f(b_touch_pos,b_touch_pos,b2_left_par,b9_touch_sens)"
    global touch_result=touch_fun_2f(b_touch_pos,b_touch_pos,b2_left_par,b9_touch_sens)
    $ 1908 "If b2_left_par"
    if (b2_left_par):
      $ 1909 "touch_result≔pose_trans(touch_result,p[-(Touch_dis)/1000,0,0,0,0,0])"
      global touch_result= pose_trans (touch_result,p[-(Touch_dis)/1000,0,0,0,0,0])
    else:
      $ 1910 "Else" "noBreak"
      $ 1911 "touch_result≔pose_trans(touch_result,p[(Touch_dis)/1000,0,0,0,0,0])"
      global touch_result= pose_trans (touch_result,p[(Touch_dis)/1000,0,0,0,0,0])
    end
    $ 1912 "A_Touch_p[A_sel_v]=touch_result"
    A_Touch_p[A_sel_v]=touch_result
    $ 1913 "If EXT_flag1[3]≟ True "
    if (EXT_flag1[3] ==   True  ):
      $ 1914 "MoveL"
      $ 1915 "manual_tp≔tilt_2f_fun(touch_result,basic_tilt_2f,wv_direction)"
      global manual_tp=tilt_2f_fun(touch_result,basic_tilt_2f,wv_direction)
      $ 1916 "manual_tp≔pose_trans(manual_tp, p[0,0,-10/1000,0,0,0])"
      global manual_tp= pose_trans (manual_tp, p[0,0,-10/1000,0,0,0])
      $ 1917 "manual_tp" "breakAfter"
      movel(pose_trans(Base, manual_tp), a=0.3, v=0.15)
      $ 1918 "Wait: 1.5"
      sleep(1.5)
    end
  end
  def MoveandTouchFun_3f():
    $ 1919 "MoveandTouchFun_3f" "noBreak"
    $ 1920 "b_touch_pos≔A_Prepos_l[A_sel_v]"
    global b_touch_pos=A_Prepos_l[A_sel_v]
    $ 1921 "tilt_deg_ry≔0"
    global tilt_deg_ry=0
    $ 1922 "tilt_deg_rz≔0"
    global tilt_deg_rz=0
    $ 1923 "If b2_left_par"
    if (b2_left_par):
      $ 1924 "tilt_deg≔6"
      global tilt_deg=6
      $ 1925 "b_touch_pos≔pose_trans(b_touch_pos, p[0,0/1000,0,d2r(tilt_deg),d2r(tilt_deg_ry),d2r(tilt_deg_rz)])"
      global b_touch_pos= pose_trans (b_touch_pos, p[0,0/1000,0,d2r(tilt_deg),d2r(tilt_deg_ry),d2r(tilt_deg_rz)])
    else:
      $ 1926 "Else" "noBreak"
      $ 1927 "tilt_deg≔0.5"
      global tilt_deg=0.5
      $ 1928 "b_touch_pos≔pose_trans(b_touch_pos, p[0,0/1000,0,d2r(-tilt_deg),d2r(tilt_deg_ry),d2r(tilt_deg_rz)])"
      global b_touch_pos= pose_trans (b_touch_pos, p[0,0/1000,0,d2r(-tilt_deg),d2r(tilt_deg_ry),d2r(tilt_deg_rz)])
    end
    $ 1939 "move_pre"
    $ 1940 "If (b2_left_par≟ True  and point_dist(A_Prepos_l[A_HOR], A_Prepos_l[A_VL1])>0.03) or (b2_left_par≟ False  and point_dist(A_Prepos_l[A_HOR_R],A_Prepos_l[A_VR1])>0.03)"
    if ((b2_left_par ==   True    and  point_dist(A_Prepos_l[A_HOR], A_Prepos_l[A_VL1])>0.03)  or  (b2_left_par ==   False    and  point_dist(A_Prepos_l[A_HOR_R],A_Prepos_l[A_VR1])>0.03)):
      $ 1941 "if move from home"
      $ 1942 "j_cp≔get_actual_joint_positions()"
      global j_cp= get_actual_joint_positions ()
      $ 1943 "If b2_left_par"
      if (b2_left_par):
        $ 1944 "If norm(b_touch_pos[1]*1000)>300"
        if (norm(b_touch_pos[1]*1000)>300):
          $ 1945 "inner_p≔p[-10/1000,-35/1000,0,0,0,0]"
          global inner_p=p[-10/1000,-35/1000,0,0,0,0]
        else:
          $ 1946 "Else" "noBreak"
          $ 1947 "inner_p≔p[0,0,0,0,0,0]"
          global inner_p=p[0,0,0,0,0,0]
        end
        $ 1948 "j_tp≔get_inverse_kin(pose_add(b_touch_pos,inner_p),qnear=left_j)"
        global j_tp= get_inverse_kin (pose_add(b_touch_pos,inner_p),qnear=left_j)
      else:
        $ 1949 "Else" "noBreak"
        $ 1950 "If norm(b_touch_pos[1]*1000)>300"
        if (norm(b_touch_pos[1]*1000)>300):
          $ 1951 "inner_p≔p[-10/1000,35/1000,0,0,0,0]"
          global inner_p=p[-10/1000,35/1000,0,0,0,0]
        else:
          $ 1952 "Else" "noBreak"
          $ 1953 "inner_p≔p[0,0,0,0,0,0]"
          global inner_p=p[0,0,0,0,0,0]
        end
        $ 1954 "j_tp≔get_inverse_kin(pose_add(b_touch_pos,inner_p),qnear=right_j)"
        global j_tp= get_inverse_kin ( pose_add (b_touch_pos,inner_p),qnear=right_j)
      end
      $ 1955 "j_cp[0]=j_tp[0]"
      j_cp[0]=j_tp[0]
      $ 1956 "j_cp[1]=j_cp[1]+(j_tp[1]-j_cp[1])/2"
      j_cp[1]=j_cp[1]+(j_tp[1]-j_cp[1])/2
      $ 1957 "j_cp[2]=j_cp[2]+(j_tp[2]-j_cp[2])/3"
      j_cp[2]=j_cp[2]+(j_tp[2]-j_cp[2])/3
      $ 1958 "j_cp[3]=j_cp[3]+(j_tp[3]-j_cp[3])/3"
      j_cp[3]=j_cp[3]+(j_tp[3]-j_cp[3])/3
      $ 1959 "j_cp[4]=j_cp[4]+(j_tp[4]-j_cp[4])/1"
      j_cp[4]=j_cp[4]+(j_tp[4]-j_cp[4])/1
      $ 1960 "j_cp[5]=j_cp[5]+(j_tp[5]-j_cp[5])/1"
      j_cp[5]=j_cp[5]+(j_tp[5]-j_cp[5])/1
      $ 1961 "MoveJ"
      $ 1962 "j_cp" "breakAfter"
      movej(j_cp, a=1.3962634015954636, v=1.0471975511965976)
      $ 1963 "j_tp≔[j_cp[0],j_cp[1],j_cp[2],j_cp[3],j_tp[4],j_tp[5]]"
      global j_tp=[j_cp[0],j_cp[1],j_cp[2],j_cp[3],j_tp[4],j_tp[5]]
      $ 1964 "MoveJ"
      $ 1965 "j_tp" "breakAfter"
      movej(j_tp, a=1.3962634015954636, v=1.0471975511965976)
    end
    $ 1966 "MoveL"
    $ 1967 "b_touch_pos" "breakAfter"
    movel(pose_trans(Base, b_touch_pos), a=0.35, v=0.35)
    $ 1970 "touch_3f_down"
    $ 1972 "touch_result≔touch_fun2(b_touch_pos,b2_left_par,b9_touch_sens,b2_par_cd)"
    global touch_result=touch_fun2(b_touch_pos,b2_left_par,b9_touch_sens,b2_par_cd)
    $ 1973 "If Scallup_check≟ False "
    if (Scallup_check ==   False  ):
      $ 1974 "touch_result≔pose_trans(touch_result,p[-(Touch_dis)/1000,0,0,0,0,0])"
      global touch_result= pose_trans (touch_result,p[-(Touch_dis)/1000,0,0,0,0,0])
    else:
      $ 1975 "Else" "noBreak"
      $ 1976 "Scallup_check≔ False "
      global Scallup_check=  False
    end
    $ 1979 "A_Touch_p[A_sel_v]=touch_result"
    A_Touch_p[A_sel_v]=touch_result
    $ 1980 "If EXT_flag1[3]≟ True "
    if (EXT_flag1[3] ==   True  ):
      $ 1981 "MoveL"
      $ 1982 "manual_tp≔tilt_3f_fun(A_Touch_p[A_sel_v],basic_tilt_3f,0)"
      global manual_tp=tilt_3f_fun(A_Touch_p[A_sel_v],basic_tilt_3f,0)
      $ 1983 "manual_tp≔pose_trans(manual_tp, p[0,0,-10/1000,0,0,0])"
      global manual_tp= pose_trans (manual_tp, p[0,0,-10/1000,0,0,0])
      $ 1984 "manual_tp" "breakAfter"
      movel(pose_trans(Base, manual_tp), a=0.3, v=0.15)
      $ 1985 "Wait: 1.5"
      sleep(1.5)
    end
    $ 1986 "touch_3f_up"
    $ 1987 "If A_Prepos_l[A_sel_v_end]≟p[0,0,0,0,0,0]"
    if (A_Prepos_l[A_sel_v_end] == p[0,0,0,0,0,0]):
      $ 1988 "A_Touch_p[A_sel_v_end]=p[0,0,0,0,0,0]"
      A_Touch_p[A_sel_v_end]=p[0,0,0,0,0,0]
    else:
      $ 1989 "Else" "noBreak"
      $ 1990 "b_touch_pos≔A_Prepos_l[A_sel_v_end]"
      global b_touch_pos=A_Prepos_l[A_sel_v_end]
      $ 1991 "MoveL"
      $ 1992 "b_touch_pos" "breakAfter"
      movel(pose_trans(Base, b_touch_pos), a=0.7, v=0.5)
      $ 1993 "touch_result≔touch_fun2(b_touch_pos,b2_left_par,b9_touch_sens)"
      global touch_result=touch_fun2(b_touch_pos,b2_left_par,b9_touch_sens)
      $ 1994 "A_Touch_p[A_sel_v_end]=touch_result"
      A_Touch_p[A_sel_v_end]=touch_result
      $ 1995 "If EXT_flag1[3]≟ True "
      if (EXT_flag1[3] ==   True  ):
        $ 1996 "MoveL"
        $ 1997 "manual_tp≔A_Touch_p[A_sel_v_end]"
        global manual_tp=A_Touch_p[A_sel_v_end]
        $ 1998 "manual_tp≔tilt_3f_fun(A_Touch_p[A_sel_v_end],basic_tilt_3f,0)"
        global manual_tp=tilt_3f_fun(A_Touch_p[A_sel_v_end],basic_tilt_3f,0)
        $ 1999 "manual_tp≔pose_trans(manual_tp, p[0,0,-10/1000,0,0,0])"
        global manual_tp= pose_trans (manual_tp, p[0,0,-10/1000,0,0,0])
        $ 2000 "manual_tp" "breakAfter"
        movel(pose_trans(Base, manual_tp), a=0.3, v=0.15)
        $ 2001 "Wait: 1.5"
        sleep(1.5)
      end
    end
  end
  def weav_welding_3f():
    $ 2005 "weav_welding_3f" "noBreak"
    $ 2006 "If running_trig≟ True "
    global thread_flag_2006=0
    thread Thread_if_2006():
      $ 2007 "inv_inching(inv_inch_time)"
      inv_inching(inv_inch_time)
      $ 2008 "b_touch_pos≔A_Prepos_l[A_sel_v]"
      global b_touch_pos=A_Prepos_l[A_sel_v]
      $ 2009 "move_pre"
      $ 2010 "j_cp≔get_actual_joint_positions()"
      global j_cp= get_actual_joint_positions ()
      $ 2011 "If b2_left_par"
      if (b2_left_par):
        $ 2012 "If norm(b_touch_pos[1]*1000)>300"
        if (norm(b_touch_pos[1]*1000)>300):
          $ 2013 "inner_p≔p[-10/1000,-35/1000,0,0,0,0]"
          global inner_p=p[-10/1000,-35/1000,0,0,0,0]
        else:
          $ 2014 "Else" "noBreak"
          $ 2015 "inner_p≔p[0,0,0,0,0,0]"
          global inner_p=p[0,0,0,0,0,0]
        end
        $ 2016 "j_tp≔get_inverse_kin(pose_add(b_touch_pos,inner_p),qnear=left_j)"
        global j_tp= get_inverse_kin (pose_add(b_touch_pos,inner_p),qnear=left_j)
      else:
        $ 2017 "Else" "noBreak"
        $ 2018 "If norm(b_touch_pos[1]*1000)>300"
        if (norm(b_touch_pos[1]*1000)>300):
          $ 2019 "inner_p≔p[-10/1000,35/1000,0,0,0,0]"
          global inner_p=p[-10/1000,35/1000,0,0,0,0]
        else:
          $ 2020 "Else" "noBreak"
          $ 2021 "inner_p≔p[0,0,0,0,0,0]"
          global inner_p=p[0,0,0,0,0,0]
        end
        $ 2022 "j_tp≔get_inverse_kin(pose_add(b_touch_pos,inner_p),qnear=right_j)"
        global j_tp= get_inverse_kin ( pose_add (b_touch_pos,inner_p),qnear=right_j)
      end
      $ 2023 "j_cp[0]=j_tp[0]"
      j_cp[0]=j_tp[0]
      $ 2024 "j_cp[1]=j_cp[1]+(j_tp[1]-j_cp[1])/2"
      j_cp[1]=j_cp[1]+(j_tp[1]-j_cp[1])/2
      $ 2025 "j_cp[2]=j_cp[2]+(j_tp[2]-j_cp[2])/3"
      j_cp[2]=j_cp[2]+(j_tp[2]-j_cp[2])/3
      $ 2026 "j_cp[3]=j_cp[3]+(j_tp[3]-j_cp[3])/3"
      j_cp[3]=j_cp[3]+(j_tp[3]-j_cp[3])/3
      $ 2027 "j_cp[4]=j_cp[4]+(j_tp[4]-j_cp[4])/1"
      j_cp[4]=j_cp[4]+(j_tp[4]-j_cp[4])/1
      $ 2028 "j_cp[5]=j_cp[5]+(j_tp[5]-j_cp[5])/1"
      j_cp[5]=j_cp[5]+(j_tp[5]-j_cp[5])/1
      $ 2029 "MoveJ"
      $ 2030 "j_cp" "breakAfter"
      movej(j_cp, a=1.3962634015954636, v=1.0471975511965976)
      $ 2031 "j_tp≔[j_cp[0],j_cp[1],j_cp[2],j_cp[3],j_tp[4],j_tp[5]]"
      global j_tp=[j_cp[0],j_cp[1],j_cp[2],j_cp[3],j_tp[4],j_tp[5]]
      $ 2032 "MoveJ"
      $ 2033 "j_tp" "breakAfter"
      movej(j_tp, a=1.3962634015954636, v=1.0471975511965976)
      $ 2034 "MoveL"
      $ 2035 "b_touch_pos" "breakAfter"
      movel(pose_trans(Base, b_touch_pos), a=0.35, v=0.35)
      $ 2036 "If (b2_left_par≟ True ) and (b1_cell_info_L≟A or b1_cell_info_L≟C or b1_cell_info_L≟c) and (A_sel_v≠A_VL2)"
      if ((b2_left_par ==   True  )  and  (b1_cell_info_L == A  or  b1_cell_info_L == C  or  b1_cell_info_L == c)  and  (A_sel_v != A_VL2)):
        $ 2037 "begin_3f_p≔pose_trans(A_Touch_p[A_sel_v],p[(multi_offset_z*(multi_path-1))/1000,0,0,0,0,0])"
        global begin_3f_p= pose_trans (A_Touch_p[A_sel_v],p[(multi_offset_z*(multi_path-1))/1000,0,0,0,0,0])
      else:
        $ 2038 "ElseIf (b2_left_par≟ False ) and (b1_cell_info_R≟A or b1_cell_info_R≟C or b1_cell_info_R≟c) and (A_sel_v≠A_VR2)"
        if ((b2_left_par ==   False  )  and  (b1_cell_info_R == A  or  b1_cell_info_R == C  or  b1_cell_info_R == c)  and  (A_sel_v != A_VR2)):
          $ 2039 "begin_3f_p≔pose_trans(A_Touch_p[A_sel_v],p[(multi_offset_z*(multi_path-1))/1000,0,0,0,0,0])"
          global begin_3f_p= pose_trans (A_Touch_p[A_sel_v],p[(multi_offset_z*(multi_path-1))/1000,0,0,0,0,0])
        else:
          $ 2040 "Else" "noBreak"
          $ 2041 "begin_3f_p≔A_Touch_p[A_sel_v]"
          global begin_3f_p=A_Touch_p[A_sel_v]
        end
      end
      $ 2042 "If b2_left_par≟ False "
      if (b2_left_par ==   False  ):
        $ 2043 "If (b1_cell_info_R≟c or b1_cell_info_R≟d) and A_sel_v≟A_VR2"
        if ((b1_cell_info_R == c  or  b1_cell_info_R == d)  and  A_sel_v == A_VR2):
          $ 2045 "b7_tilt_degree≔[-72,-20,15]"
          global b7_tilt_degree=[-72,-20,15]
          $ 2046 "begin_3f_p=pose_add(begin_3f_p,p[-6/1000,-1.5/1000,0,0,0,0])"
          begin_3f_p= pose_add (begin_3f_p,p[-6/1000,-1.5/1000,0,0,0,0])
          $ 2047 "a2_speed_cpm≔a2_speed_cpm*1"
          global a2_speed_cpm=a2_speed_cpm*1
          $ 2048 "a3_wv_amplitude≔a3_wv_amplitude*1"
          global a3_wv_amplitude=a3_wv_amplitude*1
          $ 2049 "a4_wv_frequency≔a4_wv_frequency*1"
          global a4_wv_frequency=a4_wv_frequency*1
          $ 2050 "b3_dealy_all≔[0,b4_wv_delay2*1,0,b6_wv_delay4*1]"
          global b3_dealy_all=[0,b4_wv_delay2*1,0,b6_wv_delay4*1]
          $ 2051 "a0_volt_ref≔a0_volt_ref*1"
          global a0_volt_ref=a0_volt_ref*1
          $ 2052 "a1_amp_ref≔a1_amp_ref*1"
          global a1_amp_ref=a1_amp_ref*1
          $ 2053 "volt and current"
          $ 2054 "squash_l≔[a0_volt_ref,a1_amp_ref,squash_enable,squash_voltage,squash_current,squash_amp,squash_speed,squash_cycle,waste_cycle,c0_offset_x,c0_offset_z]"
          global squash_l=[a0_volt_ref,a1_amp_ref,squash_enable,squash_voltage,squash_current,squash_amp,squash_speed,squash_cycle,waste_cycle,c0_offset_x,c0_offset_z]
          $ 2055 "set_current_voltage(a1_amp_ref,a0_volt_ref)"
          set_current_voltage(a1_amp_ref,a0_volt_ref)
        end
      end
      $ 2064 "welding_result = line_weaving_tp(begin_3f_p,A_Touch_p[A_sel_v_end],[a8_wv_distance,Circle_Speed,b1_appro_param,a4_wv_frequency,a3_wv_amplitude,b8_wv_type,wv_direction],b7_tilt_degree,b3_dealy_all,a9_wv_weldingon,c3_wv_arc,c7_wv_gap,a5_f_hole,b8_wv_2f,a7_weld_crater,squash_l)"
      welding_result = line_weaving_tp(begin_3f_p,A_Touch_p[A_sel_v_end],[a8_wv_distance,Circle_Speed,b1_appro_param,a4_wv_frequency,a3_wv_amplitude,b8_wv_type,wv_direction],b7_tilt_degree,b3_dealy_all,a9_wv_weldingon,c3_wv_arc,c7_wv_gap,a5_f_hole,b8_wv_2f,a7_weld_crater,squash_l)
      thread_flag_2006 = 1
    end
    if (running_trig ==   True  ):
      global thread_handler_2006=run Thread_if_2006()
      while (thread_flag_2006 == 0):
        if not(running_trig ==   True  ):
          kill thread_handler_2006
          thread_flag_2006 = 2
        else:
          sync()
        end
      end
    else:
      thread_flag_2006 = 2
    end
    $ 2065 "write_port_register(weld_done_137,1)"
    write_port_register(weld_done_137,1)
    $ 2066 "homeing()"
    homeing()
    $ 2067 "If sludge≟1"
    if (sludge == 1):
      $ 2068 "pause_trig≔ True "
      global pause_trig=  True
    end
  end
  def weav_welding_2f():
    $ 2069 "weav_welding_2f" "noBreak"
    $ 2070 "If running_trig≟ True "
    global thread_flag_2070=0
    thread Thread_if_2070():
      $ 2071 "Calculation"
      $ 2072 "If Auto_W_num[Auto_cur_cell]≟31 or Auto_W_num[Auto_cur_cell]≟32 or Auto_W_num[Auto_cur_cell]≟30"
      if (Auto_W_num[Auto_cur_cell] == 31  or  Auto_W_num[Auto_cur_cell] == 32  or  Auto_W_num[Auto_cur_cell] == 30):
        $ 2073 "cal_single"
        $ 2074 "pos_m_path≔A_Touch_p[A_HOR]"
        global pos_m_path=A_Touch_p[A_HOR]
        $ 2075 "pos_m_path_end≔A_Touch_p[A_HOR_R]"
        global pos_m_path_end=A_Touch_p[A_HOR_R]
        $ 2076 "A_middle_weld≔interpolate_pose(pos_m_path, pos_m_path_end,0.5)"
        global A_middle_weld= interpolate_pose (pos_m_path, pos_m_path_end,0.5)
      else:
        $ 2077 "Else" "noBreak"
        $ 2078 "side_offset≔10*current_path"
        global side_offset=10*current_path
        $ 2079 "side_offset≔0"
        global side_offset=0
        $ 2080 "If current_path≟2 or current_path≟4"
        if (current_path == 2  or  current_path == 4):
          $ 2081 "center_offset≔15"
          global center_offset=15
        else:
          $ 2082 "Else" "noBreak"
          $ 2083 "center_offset≔0"
          global center_offset=0
        end
        $ 2084 "cal_multi"
        $ 2085 "pos_m_path≔A_Touch_p[A_HOR]"
        global pos_m_path=A_Touch_p[A_HOR]
        $ 2086 "pos_m_path≔pose_trans(pos_m_path, p[side_offset/1000,0,0,0,0,0])"
        global pos_m_path= pose_trans (pos_m_path, p[side_offset/1000,0,0,0,0,0])
        $ 2087 "pos_m_path_end≔A_Touch_p[A_HOR_R]"
        global pos_m_path_end=A_Touch_p[A_HOR_R]
        $ 2088 "pos_m_path_end≔pose_trans(pos_m_path_end, p[-side_offset/1000,0,0,0,0,0])"
        global pos_m_path_end= pose_trans (pos_m_path_end, p[-side_offset/1000,0,0,0,0,0])
        $ 2089 "A_middle_weld≔interpolate_pose(pos_m_path, pos_m_path_end,0.5)"
        global A_middle_weld= interpolate_pose (pos_m_path, pos_m_path_end,0.5)
        $ 2090 "A_middle_weld≔pose_trans(A_middle_weld, p[-center_offset/1000,0,0,0,0,0])"
        global A_middle_weld= pose_trans (A_middle_weld, p[-center_offset/1000,0,0,0,0,0])
      end
      $ 2091 "gap_half"
      $ 2092 "gap_amp_bak≔c5_wv_gap_y"
      global gap_amp_bak=c5_wv_gap_y
      $ 2093 "gap_speed_bak≔c6_wv_gap_cpm"
      global gap_speed_bak=c6_wv_gap_cpm
      $ 2094 "gap_freq_bak≔c9_wv_gap_freq"
      global gap_freq_bak=c9_wv_gap_freq
      $ 2095 "c5_wv_gap_y≔(a3_wv_amplitude+c5_wv_gap_y)/2"
      global c5_wv_gap_y=(a3_wv_amplitude+c5_wv_gap_y)/2
      $ 2096 "c6_wv_gap_cpm≔(a2_speed_cpm+c6_wv_gap_cpm)/2"
      global c6_wv_gap_cpm=(a2_speed_cpm+c6_wv_gap_cpm)/2
      $ 2097 "c9_wv_gap_freq≔(a4_wv_frequency+c9_wv_gap_freq)/2"
      global c9_wv_gap_freq=(a4_wv_frequency+c9_wv_gap_freq)/2
      $ 2098 "c7_wv_gap≔[c4_gap_enable,c5_wv_gap_y,c6_wv_gap_cpm,c9_wv_gap_freq]"
      global c7_wv_gap=[c4_gap_enable,c5_wv_gap_y,c6_wv_gap_cpm,c9_wv_gap_freq]
      $ 2099 "Weaving"
      $ 2100 "If EXT_flag1[6]"
      if (EXT_flag1[6]):
        $ 2101 "If Auto_W_num[Auto_cur_cell]%10≟1"
        if (Auto_W_num[Auto_cur_cell]%10 == 1):
          $ 2102 "inv_inching(inv_inch_time)"
          inv_inching(inv_inch_time)
          $ 2103 "wv_direction≔1"
          global wv_direction=1
          $ 2104 "welding_result = line_weaving_tp(pos_m_path,A_middle_weld,[a8_wv_distance,Circle_Speed,b1_appro_param,a4_wv_frequency,a3_wv_amplitude,b8_wv_type,wv_direction],b7_tilt_degree,b3_dealy_all,a9_wv_weldingon,c3_wv_arc,c7_wv_gap,a5_f_hole,b8_wv_2f,a7_weld_crater,squash_l)"
          welding_result = line_weaving_tp(pos_m_path,A_middle_weld,[a8_wv_distance,Circle_Speed,b1_appro_param,a4_wv_frequency,a3_wv_amplitude,b8_wv_type,wv_direction],b7_tilt_degree,b3_dealy_all,a9_wv_weldingon,c3_wv_arc,c7_wv_gap,a5_f_hole,b8_wv_2f,a7_weld_crater,squash_l)
          $ 2105 "Wait: 0.5"
          sleep(0.5)
        end
        $ 2106 "If Auto_W_num[Auto_cur_cell]%10≟2"
        if (Auto_W_num[Auto_cur_cell]%10 == 2):
          $ 2107 "inv_inching(inv_inch_time)"
          inv_inching(inv_inch_time)
          $ 2108 "a7_weld_crater≔[d_start_current,d_start_voltage,d_start_time,d_end_current_2,d_end_voltage_2,d_end_time_2,d_lean_degree]"
          global a7_weld_crater=[d_start_current,d_start_voltage,d_start_time,d_end_current_2,d_end_voltage_2,d_end_time_2,d_lean_degree]
          $ 2109 "gap_half_right"
          $ 2110 "a3_wv_amplitude≔gap_amp_bak"
          global a3_wv_amplitude=gap_amp_bak
          $ 2111 "a2_speed_cpm≔gap_speed_bak"
          global a2_speed_cpm=gap_speed_bak
          $ 2112 "a4_wv_frequency≔gap_freq_bak"
          global a4_wv_frequency=gap_freq_bak
          $ 2113 "c7_wv_gap≔[c4_gap_enable,c5_wv_gap_y,c6_wv_gap_cpm,c9_wv_gap_freq]"
          global c7_wv_gap=[c4_gap_enable,c5_wv_gap_y,c6_wv_gap_cpm,c9_wv_gap_freq]
          $ 2114 "wv_direction≔-1"
          global wv_direction=-1
          $ 2115 "A_middle_weld≔feature_offset(A_middle_weld,p[-20/1000,0,0,0,0,0],A_Touch_p[A_sel_v])"
          global A_middle_weld=feature_offset(A_middle_weld,p[-20/1000,0,0,0,0,0],A_Touch_p[A_sel_v])
          $ 2116 "welding_result = line_weaving_tp(pos_m_path_end,A_middle_weld,[a8_wv_distance,Circle_Speed,b1_appro_param,a4_wv_frequency,a3_wv_amplitude,b8_wv_type,wv_direction],b7_tilt_degree,b3_dealy_all,a9_wv_weldingon,c3_wv_arc,c7_wv_gap,a5_f_hole,b8_wv_2f,a7_weld_crater,squash_l)"
          welding_result = line_weaving_tp(pos_m_path_end,A_middle_weld,[a8_wv_distance,Circle_Speed,b1_appro_param,a4_wv_frequency,a3_wv_amplitude,b8_wv_type,wv_direction],b7_tilt_degree,b3_dealy_all,a9_wv_weldingon,c3_wv_arc,c7_wv_gap,a5_f_hole,b8_wv_2f,a7_weld_crater,squash_l)
        end
      else:
        $ 2118 "Else" "noBreak"
        $ 2119 "If Auto_W_num[Auto_cur_cell]%10≟0"
        if (Auto_W_num[Auto_cur_cell]%10 == 0):
          $ 2120 "inv_inching(inv_inch_time)"
          inv_inching(inv_inch_time)
          $ 2121 "wv_direction≔1"
          global wv_direction=1
          $ 2122 "welding_result = line_weaving_tp(pos_m_path,pos_m_path_end,[a8_wv_distance,Circle_Speed,b1_appro_param,a4_wv_frequency,a3_wv_amplitude,b8_wv_type,wv_direction],b7_tilt_degree,b3_dealy_all,a9_wv_weldingon,c3_wv_arc,c7_wv_gap,a5_f_hole,b8_wv_2f,a7_weld_crater,squash_l)"
          welding_result = line_weaving_tp(pos_m_path,pos_m_path_end,[a8_wv_distance,Circle_Speed,b1_appro_param,a4_wv_frequency,a3_wv_amplitude,b8_wv_type,wv_direction],b7_tilt_degree,b3_dealy_all,a9_wv_weldingon,c3_wv_arc,c7_wv_gap,a5_f_hole,b8_wv_2f,a7_weld_crater,squash_l)
        else:
          $ 2123 "Else" "noBreak"
          $ 2124 "write_port_register(142,142)"
          write_port_register(142,142)
          $ 2125 "Halt"
          halt
        end
      end
      thread_flag_2070 = 1
    end
    if (running_trig ==   True  ):
      global thread_handler_2070=run Thread_if_2070()
      while (thread_flag_2070 == 0):
        if not(running_trig ==   True  ):
          kill thread_handler_2070
          thread_flag_2070 = 2
        else:
          sync()
        end
      end
    else:
      thread_flag_2070 = 2
    end
    $ 2126 "write_port_register(weld_done_137,1)"
    write_port_register(weld_done_137,1)
    $ 2127 "MoveL"
    $ 2128 "Direction: Tool Z-"
    global move_thread_flag_2128=0
    thread move_thread_2128():
      enter_critical
      move_thread_flag_2128 = 1
      local towardsPos=calculate_point_to_move_towards(get_forward_kin(), [0.0,0.0,-1.0], 0.03)
      movel(towardsPos, a=1.2, v=0.25)
      move_thread_flag_2128 = 2
      exit_critical
    end
    move_thread_flag_2128 = 0
    move_thread_han_2128 = run move_thread_2128()
    while (True):
      sleep(1.0E-10)
      if (move_thread_flag_2128 > 1):
        join move_thread_han_2128
        $ 2129 "Until (distance)"
        break
      end
      sync()
    end
    $ 2130 "homeing()"
    homeing()
    $ 2131 "If sludge≟1 or (sludge≟2 and current_path>1)"
    if (sludge == 1  or  (sludge == 2  and  current_path>1)):
      $ 2132 "If  not (Auto_W_num[Auto_cur_cell]%10≟1)"
      if (  not  (Auto_W_num[Auto_cur_cell]%10 == 1)):
        $ 2133 "pause_trig≔ True "
        global pause_trig=  True
      end
    end
  end
  def weav_welding_2f_CD():
    $ 2134 "weav_welding_2f_CD" "noBreak"
    $ 2135 "If running_trig≟ True "
    global thread_flag_2135=0
    thread Thread_if_2135():
      $ 2136 "CD_calculation"
      $ 2137 "If (Auto_W_num[Auto_cur_cell]≥100 and Auto_W_num[Auto_cur_cell]<106)  or (Auto_W_num[Auto_cur_cell]≥150 and Auto_W_num[Auto_cur_cell]<156)"
      if ((Auto_W_num[Auto_cur_cell] >= 100  and  Auto_W_num[Auto_cur_cell]<106)   or  (Auto_W_num[Auto_cur_cell] >= 150  and  Auto_W_num[Auto_cur_cell]<156)):
        $ 2138 "cal single"
        $ 2139 "cal_1"
        $ 2140 "pos_m_path_cd≔A_Touch_p[A_sel_v]"
        global pos_m_path_cd=A_Touch_p[A_sel_v]
        $ 2141 "pos_m_p_end_cd≔A_Touch_p[A_sel_v_end]"
        global pos_m_p_end_cd=A_Touch_p[A_sel_v_end]
        $ 2142 "cal_2"
        $ 2143 "pos_m_path≔A_Touch_p[A_sel_v2]"
        global pos_m_path=A_Touch_p[A_sel_v2]
        $ 2144 "pos_m_path_end≔A_Touch_p[A_sel_v_end2]"
        global pos_m_path_end=A_Touch_p[A_sel_v_end2]
        $ 2145 "A_middle_weld≔interpolate_pose(pos_m_path, pos_m_path_end,0.5)"
        global A_middle_weld= interpolate_pose (pos_m_path, pos_m_path_end,0.5)
      else:
        $ 2146 "Else" "noBreak"
        $ 2147 "cal multi"
        $ 2148 "side_offset≔0"
        global side_offset=0
        $ 2149 "If current_path≟2 or current_path≟4"
        if (current_path == 2  or  current_path == 4):
          $ 2150 "center_offset≔15"
          global center_offset=15
        else:
          $ 2151 "Else" "noBreak"
          $ 2152 "center_offset≔0"
          global center_offset=0
        end
        $ 2153 "cal_1_multi"
        $ 2154 "pos_m_path_cd≔A_Touch_p[A_sel_v]"
        global pos_m_path_cd=A_Touch_p[A_sel_v]
        $ 2155 "pos_m_path_cd≔pose_trans(pos_m_path_cd, p[side_offset/1000,0,0,0,0,0])"
        global pos_m_path_cd= pose_trans (pos_m_path_cd, p[side_offset/1000,0,0,0,0,0])
        $ 2156 "pos_m_p_end_cd≔A_Touch_p[A_sel_v_end]"
        global pos_m_p_end_cd=A_Touch_p[A_sel_v_end]
        $ 2157 "pos_m_p_end_cd≔pose_trans(pos_m_p_end_cd, p[-side_offset/1000,0,0,0,0,0])"
        global pos_m_p_end_cd= pose_trans (pos_m_p_end_cd, p[-side_offset/1000,0,0,0,0,0])
        $ 2158 "cal_2_multi"
        $ 2159 "pos_m_path≔A_Touch_p[A_sel_v2]"
        global pos_m_path=A_Touch_p[A_sel_v2]
        $ 2160 "pos_m_path≔pose_trans(pos_m_path, p[side_offset/1000,0,0,0,0,0])"
        global pos_m_path= pose_trans (pos_m_path, p[side_offset/1000,0,0,0,0,0])
        $ 2161 "pos_m_path_end≔A_Touch_p[A_sel_v_end2]"
        global pos_m_path_end=A_Touch_p[A_sel_v_end2]
        $ 2162 "pos_m_path_end≔pose_trans(pos_m_path_end, p[-side_offset/1000,0,0,0,0,0])"
        global pos_m_path_end= pose_trans (pos_m_path_end, p[-side_offset/1000,0,0,0,0,0])
        $ 2163 "A_middle_weld≔interpolate_pose(pos_m_path, pos_m_path_end,0.5)"
        global A_middle_weld= interpolate_pose (pos_m_path, pos_m_path_end,0.5)
        $ 2164 "A_middle_weld≔pose_trans(A_middle_weld, p[center_offset*wv_direction/1000,0,0,0,0,0])"
        global A_middle_weld= pose_trans (A_middle_weld, p[center_offset*wv_direction/1000,0,0,0,0,0])
      end
      $ 2165 "gap_half"
      $ 2166 "gap_amp_bak≔c5_wv_gap_y"
      global gap_amp_bak=c5_wv_gap_y
      $ 2167 "gap_speed_bak≔c6_wv_gap_cpm"
      global gap_speed_bak=c6_wv_gap_cpm
      $ 2168 "gap_freq_bak≔c9_wv_gap_freq"
      global gap_freq_bak=c9_wv_gap_freq
      $ 2169 "c5_wv_gap_y≔(a3_wv_amplitude+c5_wv_gap_y)/2"
      global c5_wv_gap_y=(a3_wv_amplitude+c5_wv_gap_y)/2
      $ 2170 "c6_wv_gap_cpm≔(a2_speed_cpm+c6_wv_gap_cpm)/2"
      global c6_wv_gap_cpm=(a2_speed_cpm+c6_wv_gap_cpm)/2
      $ 2171 "c9_wv_gap_freq≔(a4_wv_frequency+c9_wv_gap_freq)/2"
      global c9_wv_gap_freq=(a4_wv_frequency+c9_wv_gap_freq)/2
      $ 2172 "c7_wv_gap≔[c4_gap_enable,c5_wv_gap_y,c6_wv_gap_cpm,c9_wv_gap_freq]"
      global c7_wv_gap=[c4_gap_enable,c5_wv_gap_y,c6_wv_gap_cpm,c9_wv_gap_freq]
      $ 2173 "If EXT_flag1[4]≟ True  and (b1_cell_info_L≠c and b1_cell_info_L≠d and b1_cell_info_R≠c and b1_cell_info_R≠d)"
      if (EXT_flag1[4] ==   True    and  (b1_cell_info_L != c  and  b1_cell_info_L != d  and  b1_cell_info_R != c  and  b1_cell_info_R != d)):
        $ 2174 "If EXT_flag1[6]"
        if (EXT_flag1[6]):
          $ 2175 "If Auto_W_num[Auto_cur_cell]%10≟1"
          if (Auto_W_num[Auto_cur_cell]%10 == 1):
            $ 2176 "inv_inching(inv_inch_time)"
            inv_inching(inv_inch_time)
            $ 2177 "welding_result = line_weaving_tp_l(pos_m_path_cd,[pos_m_p_end_cd,pos_m_path,A_middle_weld],[a8_wv_distance,Circle_Speed,b1_appro_param,a4_wv_frequency,a3_wv_amplitude,b8_wv_type,wv_direction],b7_tilt_degree,b3_dealy_all,a9_wv_weldingon,c3_wv_arc,c7_wv_gap,a5_f_hole,b8_wv_2f,a7_weld_crater,squash_l)"
            welding_result = line_weaving_tp_l(pos_m_path_cd,[pos_m_p_end_cd,pos_m_path,A_middle_weld],[a8_wv_distance,Circle_Speed,b1_appro_param,a4_wv_frequency,a3_wv_amplitude,b8_wv_type,wv_direction],b7_tilt_degree,b3_dealy_all,a9_wv_weldingon,c3_wv_arc,c7_wv_gap,a5_f_hole,b8_wv_2f,a7_weld_crater,squash_l)
          end
          $ 2178 "If Auto_W_num[Auto_cur_cell]%10≟4"
          if (Auto_W_num[Auto_cur_cell]%10 == 4):
            $ 2179 "inv_inching(inv_inch_time)"
            inv_inching(inv_inch_time)
            $ 2180 "a7_weld_crater≔[d_start_current,d_start_voltage,d_start_time,d_end_current_2,d_end_voltage_2,d_end_time_2,d_lean_degree]"
            global a7_weld_crater=[d_start_current,d_start_voltage,d_start_time,d_end_current_2,d_end_voltage_2,d_end_time_2,d_lean_degree]
            $ 2181 "gap_half"
            $ 2182 "a3_wv_amplitude≔gap_amp_bak"
            global a3_wv_amplitude=gap_amp_bak
            $ 2183 "a2_speed_cpm≔gap_speed_bak"
            global a2_speed_cpm=gap_speed_bak
            $ 2184 "a4_wv_frequency≔gap_freq_bak"
            global a4_wv_frequency=gap_freq_bak
            $ 2185 "c7_wv_gap≔[c4_gap_enable,c5_wv_gap_y,c6_wv_gap_cpm,c9_wv_gap_freq]"
            global c7_wv_gap=[c4_gap_enable,c5_wv_gap_y,c6_wv_gap_cpm,c9_wv_gap_freq]
            $ 2186 "wv_direction≔-1*wv_direction"
            global wv_direction=-1*wv_direction
            $ 2187 "A_middle_weld≔feature_offset(A_middle_weld,p[20*wv_direction/1000,0,0,0,0,0],A_Touch_p[A_sel_v2])"
            global A_middle_weld=feature_offset(A_middle_weld,p[20*wv_direction/1000,0,0,0,0,0],A_Touch_p[A_sel_v2])
            $ 2188 "welding_result = line_weaving_tp(pos_m_path_end,A_middle_weld,[a8_wv_distance,Circle_Speed,b1_appro_param,a4_wv_frequency,a3_wv_amplitude,b8_wv_type,wv_direction],b7_tilt_degree,b3_dealy_all,a9_wv_weldingon,c3_wv_arc,c7_wv_gap,a5_f_hole,b8_wv_2f,a7_weld_crater,squash_l)"
            welding_result = line_weaving_tp(pos_m_path_end,A_middle_weld,[a8_wv_distance,Circle_Speed,b1_appro_param,a4_wv_frequency,a3_wv_amplitude,b8_wv_type,wv_direction],b7_tilt_degree,b3_dealy_all,a9_wv_weldingon,c3_wv_arc,c7_wv_gap,a5_f_hole,b8_wv_2f,a7_weld_crater,squash_l)
          end
        else:
          $ 2189 "Else" "noBreak"
          $ 2190 "If Auto_W_num[Auto_cur_cell]%10≟0"
          if (Auto_W_num[Auto_cur_cell]%10 == 0):
            $ 2191 "inv_inching(inv_inch_time)"
            inv_inching(inv_inch_time)
            $ 2192 "welding_result = line_weaving_tp_l(pos_m_path_cd,[pos_m_p_end_cd,pos_m_path,pos_m_path_end],[a8_wv_distance,Circle_Speed,b1_appro_param,a4_wv_frequency,a3_wv_amplitude,b8_wv_type,wv_direction],b7_tilt_degree,b3_dealy_all,a9_wv_weldingon,c3_wv_arc,c7_wv_gap,a5_f_hole,b8_wv_2f,a7_weld_crater,squash_l)"
            welding_result = line_weaving_tp_l(pos_m_path_cd,[pos_m_p_end_cd,pos_m_path,pos_m_path_end],[a8_wv_distance,Circle_Speed,b1_appro_param,a4_wv_frequency,a3_wv_amplitude,b8_wv_type,wv_direction],b7_tilt_degree,b3_dealy_all,a9_wv_weldingon,c3_wv_arc,c7_wv_gap,a5_f_hole,b8_wv_2f,a7_weld_crater,squash_l)
          else:
            $ 2193 "Else" "noBreak"
            $ 2194 "write_port_register(142,142)"
            write_port_register(142,142)
            $ 2195 "Halt"
            halt
          end
        end
      else:
        $ 2196 "Else" "noBreak"
        $ 2197 "If EXT_flag1[6]"
        if (EXT_flag1[6]):
          $ 2198 "If Auto_W_num[Auto_cur_cell]%10≟2"
          if (Auto_W_num[Auto_cur_cell]%10 == 2):
            $ 2199 "inv_inching(inv_inch_time)"
            inv_inching(inv_inch_time)
            $ 2200 "gap_half"
            $ 2201 "gap_amp_bak≔c5_wv_gap_y"
            global gap_amp_bak=c5_wv_gap_y
            $ 2202 "gap_speed_bak≔c6_wv_gap_cpm"
            global gap_speed_bak=c6_wv_gap_cpm
            $ 2203 "gap_freq_bak≔c9_wv_gap_freq"
            global gap_freq_bak=c9_wv_gap_freq
            $ 2204 "c5_wv_gap_y≔(a3_wv_amplitude+c5_wv_gap_y)/2"
            global c5_wv_gap_y=(a3_wv_amplitude+c5_wv_gap_y)/2
            $ 2205 "c6_wv_gap_cpm≔(a2_speed_cpm+c6_wv_gap_cpm)/2"
            global c6_wv_gap_cpm=(a2_speed_cpm+c6_wv_gap_cpm)/2
            $ 2206 "c9_wv_gap_freq≔(a4_wv_frequency+c9_wv_gap_freq)/2"
            global c9_wv_gap_freq=(a4_wv_frequency+c9_wv_gap_freq)/2
            $ 2207 "c7_wv_gap≔[c4_gap_enable,c5_wv_gap_y,c6_wv_gap_cpm,c9_wv_gap_freq]"
            global c7_wv_gap=[c4_gap_enable,c5_wv_gap_y,c6_wv_gap_cpm,c9_wv_gap_freq]
            $ 2208 "welding_result = line_weaving_tp(pos_m_path_cd,pos_m_p_end_cd,[a8_wv_distance,Circle_Speed,b1_appro_param,a4_wv_frequency,a3_wv_amplitude,b8_wv_type,wv_direction],b7_tilt_degree,b3_dealy_all,a9_wv_weldingon,c3_wv_arc,c7_wv_gap,a5_f_hole,b8_wv_2f,a7_weld_crater,squash_l)"
            welding_result = line_weaving_tp(pos_m_path_cd,pos_m_p_end_cd,[a8_wv_distance,Circle_Speed,b1_appro_param,a4_wv_frequency,a3_wv_amplitude,b8_wv_type,wv_direction],b7_tilt_degree,b3_dealy_all,a9_wv_weldingon,c3_wv_arc,c7_wv_gap,a5_f_hole,b8_wv_2f,a7_weld_crater,squash_l)
            $ 2209 "Wait: 0.5"
            sleep(0.5)
          end
          $ 2210 "If Auto_W_num[Auto_cur_cell]%10≟3"
          if (Auto_W_num[Auto_cur_cell]%10 == 3):
            $ 2211 "inv_inching(inv_inch_time)"
            inv_inching(inv_inch_time)
            $ 2212 "welding_result = line_weaving_tp(pos_m_path,A_middle_weld,[a8_wv_distance,Circle_Speed,b1_appro_param,a4_wv_frequency,a3_wv_amplitude,b8_wv_type,wv_direction],b7_tilt_degree,b3_dealy_all,a9_wv_weldingon,c3_wv_arc,c7_wv_gap,a5_f_hole,b8_wv_2f,a7_weld_crater,squash_l)"
            welding_result = line_weaving_tp(pos_m_path,A_middle_weld,[a8_wv_distance,Circle_Speed,b1_appro_param,a4_wv_frequency,a3_wv_amplitude,b8_wv_type,wv_direction],b7_tilt_degree,b3_dealy_all,a9_wv_weldingon,c3_wv_arc,c7_wv_gap,a5_f_hole,b8_wv_2f,a7_weld_crater,squash_l)
            $ 2213 "Wait: 0.5"
            sleep(0.5)
          end
          $ 2214 "If Auto_W_num[Auto_cur_cell]%10≟4"
          if (Auto_W_num[Auto_cur_cell]%10 == 4):
            $ 2215 "inv_inching(inv_inch_time)"
            inv_inching(inv_inch_time)
            $ 2216 "a7_weld_crater≔[d_start_current,d_start_voltage,d_start_time,d_end_current_2,d_end_voltage_2,d_end_time_2,d_lean_degree]"
            global a7_weld_crater=[d_start_current,d_start_voltage,d_start_time,d_end_current_2,d_end_voltage_2,d_end_time_2,d_lean_degree]
            $ 2217 "gap_half"
            $ 2218 "a3_wv_amplitude≔gap_amp_bak"
            global a3_wv_amplitude=gap_amp_bak
            $ 2219 "a2_speed_cpm≔gap_speed_bak"
            global a2_speed_cpm=gap_speed_bak
            $ 2220 "a4_wv_frequency≔gap_freq_bak"
            global a4_wv_frequency=gap_freq_bak
            $ 2221 "c7_wv_gap≔[c4_gap_enable,c5_wv_gap_y,c6_wv_gap_cpm,c9_wv_gap_freq]"
            global c7_wv_gap=[c4_gap_enable,c5_wv_gap_y,c6_wv_gap_cpm,c9_wv_gap_freq]
            $ 2222 "wv_direction≔-1*wv_direction"
            global wv_direction=-1*wv_direction
            $ 2223 "A_middle_weld≔feature_offset(A_middle_weld,p[20*wv_direction/1000,0,0,0,0,0],A_Touch_p[A_sel_v2])"
            global A_middle_weld=feature_offset(A_middle_weld,p[20*wv_direction/1000,0,0,0,0,0],A_Touch_p[A_sel_v2])
            $ 2224 "welding_result = line_weaving_tp(pos_m_path_end,A_middle_weld,[a8_wv_distance,Circle_Speed,b1_appro_param,a4_wv_frequency,a3_wv_amplitude,b8_wv_type,wv_direction],b7_tilt_degree,b3_dealy_all,a9_wv_weldingon,c3_wv_arc,c7_wv_gap,a5_f_hole,b8_wv_2f,a7_weld_crater,squash_l)"
            welding_result = line_weaving_tp(pos_m_path_end,A_middle_weld,[a8_wv_distance,Circle_Speed,b1_appro_param,a4_wv_frequency,a3_wv_amplitude,b8_wv_type,wv_direction],b7_tilt_degree,b3_dealy_all,a9_wv_weldingon,c3_wv_arc,c7_wv_gap,a5_f_hole,b8_wv_2f,a7_weld_crater,squash_l)
          end
        else:
          $ 2225 "Else" "noBreak"
          $ 2226 "If Auto_W_num[Auto_cur_cell]%10≟2"
          if (Auto_W_num[Auto_cur_cell]%10 == 2):
            $ 2227 "inv_inching(inv_inch_time)"
            inv_inching(inv_inch_time)
            $ 2228 "c7_wv_gap≔[0,c5_wv_gap_y,c6_wv_gap_cpm,c9_wv_gap_freq]"
            global c7_wv_gap=[0,c5_wv_gap_y,c6_wv_gap_cpm,c9_wv_gap_freq]
            $ 2229 "welding_result = line_weaving_tp(pos_m_path_cd,pos_m_p_end_cd,[a8_wv_distance,Circle_Speed,b1_appro_param,a4_wv_frequency,a3_wv_amplitude,b8_wv_type,wv_direction],b7_tilt_degree,b3_dealy_all,a9_wv_weldingon,c3_wv_arc,c7_wv_gap,a5_f_hole,b8_wv_2f,a7_weld_crater,squash_l)"
            welding_result = line_weaving_tp(pos_m_path_cd,pos_m_p_end_cd,[a8_wv_distance,Circle_Speed,b1_appro_param,a4_wv_frequency,a3_wv_amplitude,b8_wv_type,wv_direction],b7_tilt_degree,b3_dealy_all,a9_wv_weldingon,c3_wv_arc,c7_wv_gap,a5_f_hole,b8_wv_2f,a7_weld_crater,squash_l)
            $ 2230 "Wait: 0.5"
            sleep(0.5)
          end
          $ 2231 "If Auto_W_num[Auto_cur_cell]%10≟5"
          if (Auto_W_num[Auto_cur_cell]%10 == 5):
            $ 2232 "inv_inching(inv_inch_time)"
            inv_inching(inv_inch_time)
            $ 2233 "c7_wv_gap≔[c4_gap_enable,c5_wv_gap_y,c6_wv_gap_cpm,c9_wv_gap_freq]"
            global c7_wv_gap=[c4_gap_enable,c5_wv_gap_y,c6_wv_gap_cpm,c9_wv_gap_freq]
            $ 2234 "welding_result = line_weaving_tp(pos_m_path,pos_m_path_end,[a8_wv_distance,Circle_Speed,b1_appro_param,a4_wv_frequency,a3_wv_amplitude,b8_wv_type,wv_direction],b7_tilt_degree,b3_dealy_all,a9_wv_weldingon,c3_wv_arc,c7_wv_gap,a5_f_hole,b8_wv_2f,a7_weld_crater,squash_l)"
            welding_result = line_weaving_tp(pos_m_path,pos_m_path_end,[a8_wv_distance,Circle_Speed,b1_appro_param,a4_wv_frequency,a3_wv_amplitude,b8_wv_type,wv_direction],b7_tilt_degree,b3_dealy_all,a9_wv_weldingon,c3_wv_arc,c7_wv_gap,a5_f_hole,b8_wv_2f,a7_weld_crater,squash_l)
            $ 2235 "Wait: 0.5"
            sleep(0.5)
          end
        end
      end
      thread_flag_2135 = 1
    end
    if (running_trig ==   True  ):
      global thread_handler_2135=run Thread_if_2135()
      while (thread_flag_2135 == 0):
        if not(running_trig ==   True  ):
          kill thread_handler_2135
          thread_flag_2135 = 2
        else:
          sync()
        end
      end
    else:
      thread_flag_2135 = 2
    end
    $ 2236 "write_port_register(weld_done_137,1)"
    write_port_register(weld_done_137,1)
    $ 2240 "wv_direction≔1"
    global wv_direction=1
    $ 2241 "If Auto_W_num[Auto_cur_cell]≥150"
    if (Auto_W_num[Auto_cur_cell] >= 150):
      $ 2242 "MoveL"
      $ 2243 "Direction: Base"
      global move_thread_flag_2243=0
      thread move_thread_2243():
        enter_critical
        move_thread_flag_2243 = 1
        local towardsPos=calculate_point_to_move_towards(p[0.0,0.0,0.0,0.0,0.0,0.0], [-1,1,0.0], 0.03)
        movel(towardsPos, a=0.2, v=0.05)
        move_thread_flag_2243 = 2
        exit_critical
      end
      move_thread_flag_2243 = 0
      move_thread_han_2243 = run move_thread_2243()
      while (True):
        sleep(1.0E-10)
        if (move_thread_flag_2243 > 1):
          join move_thread_han_2243
          $ 2244 "Until (distance)"
          break
        end
        sync()
      end
    else:
      $ 2245 "ElseIf Auto_W_num[Auto_cur_cell]≥100"
      if (Auto_W_num[Auto_cur_cell] >= 100):
        $ 2246 "MoveL"
        $ 2247 "Direction: Base"
        global move_thread_flag_2247=0
        thread move_thread_2247():
          enter_critical
          move_thread_flag_2247 = 1
          local towardsPos=calculate_point_to_move_towards(p[0.0,0.0,0.0,0.0,0.0,0.0], [-1,-1,0.0], 0.03)
          movel(towardsPos, a=0.2, v=0.05)
          move_thread_flag_2247 = 2
          exit_critical
        end
        move_thread_flag_2247 = 0
        move_thread_han_2247 = run move_thread_2247()
        while (True):
          sleep(1.0E-10)
          if (move_thread_flag_2247 > 1):
            join move_thread_han_2247
            $ 2248 "Until (distance)"
            break
          end
          sync()
        end
      end
    end
    $ 2249 "MoveL"
    $ 2250 "Direction: Tool Z-"
    global move_thread_flag_2250=0
    thread move_thread_2250():
      enter_critical
      move_thread_flag_2250 = 1
      local towardsPos=calculate_point_to_move_towards(get_forward_kin(), [0.0,0.0,-1.0], 0.03)
      movel(towardsPos, a=1.2, v=0.25)
      move_thread_flag_2250 = 2
      exit_critical
    end
    move_thread_flag_2250 = 0
    move_thread_han_2250 = run move_thread_2250()
    while (True):
      sleep(1.0E-10)
      if (move_thread_flag_2250 > 1):
        join move_thread_han_2250
        $ 2251 "Until (distance)"
        break
      end
      sync()
    end
    $ 2252 "homeing()"
    homeing()
    $ 2253 "If sludge≟1 or (sludge≟2 and current_path>1)"
    if (sludge == 1  or  (sludge == 2  and  current_path>1)):
      $ 2254 "If  not (Auto_W_num[Auto_cur_cell]%10≟1 or Auto_W_num[Auto_cur_cell]%10≟2 or Auto_W_num[Auto_cur_cell]%10≟3)"
      if (  not  (Auto_W_num[Auto_cur_cell]%10 == 1  or  Auto_W_num[Auto_cur_cell]%10 == 2  or  Auto_W_num[Auto_cur_cell]%10 == 3)):
        $ 2255 "pause_trig≔ True "
        global pause_trig=  True
      end
    end
  end
  def reset_weld_param():
    $ 2256 "reset_weld_param" "noBreak"
    $ 2257 "start_num≔225"
    global start_num=225
    $ 2258 "Loop start_num<237"
    while (start_num<237):
      $ 2259 "write_port_register(start_num,0)"
      write_port_register(start_num,0)
      $ 2260 "start_num≔start_num+1"
      global start_num=start_num+1
    end
    $ 2261 "start_num≔240"
    global start_num=240
    $ 2262 "Loop start_num<256"
    while (start_num<256):
      $ 2263 "write_port_register(start_num,0)"
      write_port_register(start_num,0)
      $ 2264 "start_num≔start_num+1"
      global start_num=start_num+1
    end
  end
  def touch_sub():
    $ 2265 "touch_sub" "noBreak"
    $ 2266 "freedrive"
    $ 2267 "save_timer: Start"
    save_timer_is_counting = True
    $ 2268 "Loop save_tool≟ False  and save_timer≤0.5"
    while (get_tool_digital_in(0) ==   False    and  save_timer <= 0.5):
      $ 2269 "If save_tool≟ False "
      if (get_tool_digital_in(0) ==   False  ):
        $ 2270 "save_timer≔0"
        global save_timer=0
      end
      $ 2271 "If freedrive≟ True  and freedrive_trg≟ False "
      if (get_tool_digital_in(1) ==   True    and  freedrive_trg ==   False  ):
        $ 2272 "'Manual - Freedrive'"
        # 'Manual - Freedrive'
        $ 2273 "freedrive_mode()"
        freedrive_mode()
        $ 2274 "freedrive_trg≔ True "
        global freedrive_trg=  True
      else:
        $ 2275 "ElseIf freedrive≟ False  and freedrive_trg≟ True "
        if (get_tool_digital_in(1) ==   False    and  freedrive_trg ==   True  ):
          $ 2276 "end_freedrive_mode()"
          end_freedrive_mode()
          $ 2277 "freedrive_trg≔ False "
          global freedrive_trg=  False
        end
      end
      $ 2278 "If lamp_trig≟ False "
      if (lamp_trig ==   False  ):
        $ 2279 "lamp_trig≔ True "
        global lamp_trig=  True
      end
      $ 2280 "sync()"
      sync()
    end
    $ 2281 "save_timer: Stop"
    save_timer_is_counting = False
    $ 2282 "save_timer: Reset"
    save_timer = 0
    $ 2283 "write_port_register(touch_done_157,1)"
    write_port_register(touch_done_157,1)
    $ 2284 "Wait read_port_register(touch_done_157)≟0"
    while (not( read_port_register (touch_done_157) == 0)):
      sync()
    end
    $ 2285 "Wait save_tool=LO"
    while (get_tool_digital_in(0) == True):
      sync()
    end
  end
  $ 2 "BeforeStart"
  $ 3 "'RobotVersion'"
  # 'RobotVersion'
  $ 4 "write_port_register(160,46)"
  write_port_register(160,46)
  $ 5 "Teaching for Touch"
  $ 6 "g_current_p≔get_actual_tcp_pose()"
  global g_current_p= get_actual_tcp_pose ()
  $ 7 "MoveJ"
  $ 8 "g_current_p" "breakAfter"
  movej(g_current_p, a=1.3962634015954636, v=1.0471975511965976, r=0.05)
  $ 9 "If  False "
  if (  False  ):
    $ 10 "MoveJ"
    $ 11 "'Home'"
    # 'Home'
    $ 12 "first_p" "breakAfter"
    movej([0.6572912931442261, -1.1853707472430628, -1.1612256209002894, -2.29183799425234, 1.5053011178970337, 2.249363422393799], a=1.3962634015954636, v=1.0471975511965976)
    $ 13 "'3F Left Right'"
    # '3F Left Right'
    $ 14 "left" "breakAfter"
    movej([1.0434843552115187, -1.5100991608390455, -1.7306758129700324, -1.1948061631169296, 1.4628666284450171, 1.848321797880608], a=1.3962634015954636, v=1.0471975511965976)
    $ 15 "right" "breakAfter"
    movej([-0.10351455753530914, -1.3302576856500608, -2.115934992292752, -0.862193753976749, 1.3219395896157813, 2.4264792168573246], a=1.3962634015954636, v=1.0471975511965976)
    $ 16 "'2F Left Right'"
    # '2F Left Right'
    $ 17 "up_left" "breakAfter"
    movej([1.1752926889699076, -1.8019900427886952, -1.320977727654376, -1.5255442863405975, 1.3476341406937622, 2.041365262351603], a=1.3962634015954636, v=1.0471975511965976)
    $ 18 "up_right" "breakAfter"
    movej([-0.490858516659304, -1.5854285429454542, -1.6450882962874376, -1.2830655228732084, 1.6157391701919699, 1.9100727821897805], a=1.3962634015954636, v=1.0471975511965976)
    $ 19 "Packing_pos" "breakAfter"
    movej([1.5877798795700073, -0.0173419157611292, -2.4983108679400843, -1.4065726439105433, 1.626846194267273, 3.0169763565063477], a=1.3962634015954636, v=1.0471975511965976)
    $ 20 "pre_position" "breakAfter"
    movej([1.2637099027633667, -0.695505444203512, -2.0481718222247522, -1.9413569609271448, 2.573765277862549, 1.3775802850723267], a=1.3962634015954636, v=1.0471975511965976)
    $ 21 "middle_pos" "breakAfter"
    movej([-1.8762093791333925, -1.0408674059020342, -1.3551139327963426, -1.843592441478755, 1.9056326083560464, 0.7075109167810423], a=1.3962634015954636, v=1.0471975511965976)
    $ 22 "Mounting_pos" "breakAfter"
    movej([0.6231353085164267, -0.6300961531972575, -0.9034285948871803, -1.770059340221131, 1.417516049558281, 1.7792033261567348], a=1.3962634015954636, v=1.0471975511965976)
    $ 23 "pre_mounting" "breakAfter"
    movej([1.2356762886047363, -0.8703244368182581, -0.942230526600973, -2.3905327955829065, 1.3216267824172974, 2.6514604091644287], a=1.3962634015954636, v=1.0471975511965976)
    $ 24 "'firstly touch center and side, side_L is side touch pose'"
    # 'firstly touch center and side, side_L is side touch pose'
    $ 25 "side_p_L" "breakAfter"
    movej([0.7063748268745771, -1.3604975314992132, -1.990433834727808, -1.0668367667667118, 1.6921872781537495, 1.2509236145111355], a=1.3962634015954636, v=1.0471975511965976)
    $ 26 "side_p_R" "breakAfter"
    movej([0.05431400611996651, -1.4896310011493128, -1.8839471975909632, -1.079590145741598, 1.21127450466156, 2.729013204574585], a=1.3962634015954636, v=1.0471975511965976)
    $ 27 "top_right" "breakAfter"
    movej([-0.02242371234582219, -0.9682979219978707, -1.1486403794481532, -1.814672356578109, 1.0564512116488283, 1.9516847799391646], a=1.3962634015954636, v=1.0471975511965976)
    $ 28 "down_right" "breakAfter"
    movej([-0.10387097169690396, -0.8634965401570085, -1.6224404602167288, -1.9527388322769834, 1.2604034373302166, 1.9362943911099855], a=1.3962634015954636, v=1.0471975511965976)
    $ 29 "way_600_3F_VL1" "breakAfter"
    movej([1.4495428629911409, -0.8691188832486789, -1.6280015865128723, -1.109862842185814, 0.958613460846621, 1.8600136596738885], a=1.3962634015954636, v=1.0471975511965976)
    $ 30 "way_3F_42" "breakAfter"
    movej([0.36805654405146704, -0.7862968504575107, -2.173257016154224, -1.4479178800416523, 0.8821879504915225, 2.8855763836420314], a=1.3962634015954636, v=1.0471975511965976)
    $ 31 "Waypoint_3" "breakAfter"
    movej([1.1380372507706311, -0.9407851141189099, -1.233329099346161, -2.2390373632318763, 1.2601061328687342, 1.8320151492624872], a=1.3962634015954636, v=1.0471975511965976)
  end
  $ 32 "waypoint"
  $ 33 "first_p_wp≔first_p"
  global first_p_wp=p[.431245807847, -.007259877891, .087796870964, 2.814824648791, -.024151220978, 1.380109909682]
  $ 34 "home_pos_j≔get_inverse_kin(first_p,qnear=[0.788235068321228, -1.101443115864889, -1.2219904104815882, -2.3243168036090296, 1.506469488143921, 2.3651483058929443])"
  global home_pos_j= get_inverse_kin (p[.431245807847, -.007259877891, .087796870964, 2.814824648791, -.024151220978, 1.380109909682],qnear=[0.788235068321228, -1.101443115864889, -1.2219904104815882, -2.3243168036090296, 1.506469488143921, 2.3651483058929443])
  $ 35 "left_j≔get_inverse_kin(left,qnear=[1.0260889556530308, -1.5106289215345097, -1.741216762689402, -1.178962336228949, 1.4987324920877318, 1.8103628938054515])"
  global left_j= get_inverse_kin (p[.480496318984, .411279115151, .006998291210, -2.211681476386, -.899147924387, -1.383032568605],qnear=[1.0260889556530308, -1.5106289215345097, -1.741216762689402, -1.178962336228949, 1.4987324920877318, 1.8103628938054515])
  $ 36 "right_j≔get_inverse_kin(right,qnear=[-0.04005625546610858, -1.5553040811514833, -1.9086689348599588, -0.877043115030812, 1.298887151057777, 2.511237649551841])"
  global right_j= get_inverse_kin (p[.475000000000, -.421403215678, .026417194146, 1.917761036827, -1.141682393512, 1.523356199292],qnear=[-0.04005625546610858, -1.5553040811514833, -1.9086689348599588, -0.877043115030812, 1.298887151057777, 2.511237649551841])
  $ 37 "Packing_pos_wp≔Packing_pos"
  global Packing_pos_wp=p[.278714911898, .357008020042, .025408199530, -2.146966801259, .195978635494, -.919933898512]
  $ 38 "pre_position_wp≔pre_position"
  global pre_position_wp=p[-.206981089246, .377817475970, .184983176991, -1.570600793609, -.863923490888, -.089005332274]
  $ 39 "pre_mounting_wp≔pre_mounting"
  global pre_mounting_wp=p[.460443249232, .114922015113, .277198878359, -2.240057458299, .067416497001, -1.614091004704]
  $ 40 "mounting_wp≔Mounting_pos"
  global mounting_wp=p[.365658114054, -.003207132620, .718667154922, -1.220752075696, -.066673751622, -2.363385143972]
  $ 41 "Setting"
  $ 42 "inv_inch_time≔0.4"
  global inv_inch_time=0.4
  $ 43 "a7_cell_bottom≔-50.2"
  global a7_cell_bottom=-50.2
  $ 44 "get_center≔470"
  global get_center=470
  $ 45 "work_touch_dis≔50"
  global work_touch_dis=50
  $ 46 "cd_extra_dis≔6"
  global cd_extra_dis=6
  $ 47 "side_pos_x≔-10"
  global side_pos_x=-10
  $ 48 "sec_touch_dis≔35"
  global sec_touch_dis=35
  $ 49 "Touch_dis≔30"
  global Touch_dis=30
  $ 50 "offset_2f_begin≔5"
  global offset_2f_begin=5
  $ 51 "offset_3f_begin≔5"
  global offset_3f_begin=5
  $ 52 "multi_offset_z≔3"
  global multi_offset_z=3
  $ 53 "simulation_mode≔ False "
  global simulation_mode=  False
  $ 54 "tilt_deg_man≔7"
  global tilt_deg_man=7
  $ 55 "Initialization"
  $ 56 "reset_revolution_counter()"
  reset_revolution_counter()
  $ 57 "get_center_bak≔get_center"
  global get_center_bak=get_center
  $ 58 "welding_program≔ False "
  global welding_program=  False
  $ 59 "vr2_p1≔p[0,0,0,0,0,0]"
  global vr2_p1=p[0,0,0,0,0,0]
  $ 60 "running_trig≔ False "
  global running_trig=  False
  $ 61 "pb_comm_count≔0"
  global pb_comm_count=0
  $ 62 "pendant_hb≔read_port_register(161)"
  global pendant_hb= read_port_register (161)
  $ 63 "pause_trig≔ False "
  global pause_trig=  False
  $ 64 "multi_path≔1"
  global multi_path=1
  $ 65 "reset_trig≔ False "
  global reset_trig=  False
  $ 66 "heartbeat≔0"
  global heartbeat=0
  $ 67 "back_2f≔ False "
  global back_2f=  False
  $ 68 "t_time≔0"
  global t_time=0
  $ 69 "cd_offset≔35"
  global cd_offset=35
  $ 70 "write_port_register(144,0)"
  write_port_register(144,0)
  $ 71 "time_cal_trig≔ False "
  global time_cal_trig=  False
  $ 72 "current_2f≔0"
  global current_2f=0
  $ 73 "A_cur_2f≔0"
  global A_cur_2f=0
  $ 74 "CD_MLR≔ True "
  global CD_MLR=  True
  $ 75 "auto_on≔ False "
  global auto_on=  False
  $ 76 "event_cal_on≔ False "
  global event_cal_on=  False
  $ 77 "event_side_on≔ False "
  global event_side_on=  False
  $ 78 "Auto_trig≔ False "
  global Auto_trig=  False
  $ 79 "lamp_trig≔ False "
  global lamp_trig=  False
  $ 80 "calcu_trig≔ False "
  global calcu_trig=  False
  $ 81 "current_path≔1"
  global current_path=1
  $ 82 "freedrive_trg≔ False "
  global freedrive_trg=  False
  $ 83 "Inch_trg≔ False "
  global Inch_trg=  False
  $ 84 "wv_direction≔1"
  global wv_direction=1
  $ 85 "Move_trig≔ False "
  global Move_trig=  False
  $ 86 "CELL_ROBOT_DIST≔500"
  global CELL_ROBOT_DIST=500
  $ 87 "CELL_WIDTH≔700"
  global CELL_WIDTH=700
  $ 88 "CELL_BOTTOM≔a7_cell_bottom"
  global CELL_BOTTOM=a7_cell_bottom
  $ 89 "scallop_info≔ False "
  global scallop_info=  False
  $ 90 "Carl_info≔ False "
  global Carl_info=  False
  $ 91 "touch_done_2f≔ False "
  global touch_done_2f=  False
  $ 92 "get_pose_side≔0"
  global get_pose_side=0
  $ 93 "get_pose_side_t≔0"
  global get_pose_side_t=0
  $ 94 "ba_trig≔ False "
  global ba_trig=  False
  $ 95 "touch_m_check≔0"
  global touch_m_check=0
  $ 96 "basic_tilt_2f≔[30,5,0]"
  global basic_tilt_2f=[30,5,0]
  $ 98 "basic_tilt_3f≔[0,-27,0]"
  global basic_tilt_3f=[0,-27,0]
  $ 100 "modbus_name"
  $ 101 "weld_done_137≔137"
  global weld_done_137=137
  $ 102 "robot_ready_141≔141"
  global robot_ready_141=141
  $ 103 "cell_3f_2f_151≔151"
  global cell_3f_2f_151=151
  $ 104 "cell_info_152≔152"
  global cell_info_152=152
  $ 105 "weld_req_153≔153"
  global weld_req_153=153
  $ 106 "touch_cell_155≔155"
  global touch_cell_155=155
  $ 107 "touch_num_156≔156"
  global touch_num_156=156
  $ 108 "touch_done_157≔157"
  global touch_done_157=157
  $ 109 "robot_move_163≔163"
  global robot_move_163=163
  $ 110 "robot_pose_164≔164"
  global robot_pose_164=164
  $ 111 "work_type_165≔165"
  global work_type_165=165
  $ 112 "arc_onoff_168≔168"
  global arc_onoff_168=168
  $ 113 "beforeafter_170≔170"
  global beforeafter_170=170
  $ 114 "return_done_240≔240"
  global return_done_240=240
  $ 115 "a0_Job_Mode≔0"
  global a0_Job_Mode=0
  $ 116 "position_3F≔1"
  global position_3F=1
  $ 117 "position_2F≔2"
  global position_2F=2
  $ 118 "cell_par"
  $ 119 "A≔1"
  global A=1
  $ 120 "B≔2"
  global B=2
  $ 121 "C≔3"
  global C=3
  $ 122 "c≔4"
  global c=4
  $ 123 "D≔5"
  global D=5
  $ 124 "d≔6"
  global d=6
  $ 125 "E≔7"
  global E=7
  $ 126 "e≔8"
  global e=8
  $ 127 "A_VL1≔1"
  global A_VL1=1
  $ 128 "A_VL2≔2"
  global A_VL2=2
  $ 129 "A_VR1≔3"
  global A_VR1=3
  $ 130 "A_VR2≔4"
  global A_VR2=4
  $ 131 "A_HOR≔5"
  global A_HOR=5
  $ 132 "A_HOR_R≔7"
  global A_HOR_R=7
  $ 133 "A_HOR_ML≔6"
  global A_HOR_ML=6
  $ 134 "A_HOR_MR≔8"
  global A_HOR_MR=8
  $ 135 "A_HOR_M≔9"
  global A_HOR_M=9
  $ 136 "A_VL1_END≔10"
  global A_VL1_END=10
  $ 137 "A_VL2_END≔11"
  global A_VL2_END=11
  $ 138 "A_VR1_END≔12"
  global A_VR1_END=12
  $ 139 "A_VR2_END≔13"
  global A_VR2_END=13
  $ 140 "A_HOR_2path≔14"
  global A_HOR_2path=14
  $ 141 "A_HOR_3path≔15"
  global A_HOR_3path=15
  $ 142 "A_HOR_4path≔16"
  global A_HOR_4path=16
  $ 143 "A_HOR_2path_CD≔17"
  global A_HOR_2path_CD=17
  $ 144 "A_HOR_3path_CD≔18"
  global A_HOR_3path_CD=18
  $ 145 "A_HOR_4path_CD≔19"
  global A_HOR_4path_CD=19
  $ 146 "Script: UR_samho_weaving_V6.8_CB.script"
  wv_wp1 = p[0,0,0,0,0,0]
  dumy_p = p[0,0,0,0,0,0]
  global background_cal = 0
  global background_pose = [dumy_p,dumy_p,dumy_p]
  global background_ready = 0
  global timer_counter = 0
  global timer_counting = False
  global wcr_counter = 0
  global wcr_counting = False
  global get_wcr = False
  global arc_sens_onoff = 0
  global welding_off_t = 55
  global weld_onoff = False
  global isHicomm = True
  global isTouchWCR = True
  global welding_program = False
  global arc_sens_2F = False

  thread thread_timer():
    error_time = 5
    start_gas_time = 2
    while (True):
      if (timer_counting):
        timer_counter = timer_counter + get_steptime()
        write_output_float_register(0,timer_counter)

        get_wcr = read_welder(5)
        weld_onoff = read_welder_control(0)

        welding_off_t = read_port_register(168)
        if(get_wcr):
          global arc_sens_onoff = 1
        else:
          global arc_sens_onoff = 0
        end
        if(get_wcr and welding_off_t == 2 and weld_onoff == True):
          wcr_counter=0
        elif(wcr_counter>(error_time+start_gas_time) and welding_off_t == 2 and weld_onoff == True):
          write_port_register(202,0)
          write_port_register(149,0)
          write_welder(0,False)
          set_standard_digital_out(0,False)
          write_port_register(142,131)
          sleep(0.5)
          halt
        elif(get_wcr == False and welding_off_t == 2 and weld_onoff == True):
          wcr_counter = wcr_counter + get_steptime()
        end
      end
      sync()
    end
  end

  def RTDE_init():
    # timer
    write_output_float_register(0,0)
    # WCR IN
    write_output_float_register(1,0)
    # Welding Current
    write_output_float_register(2,0)
    # Welding Voltage
    write_output_float_register(3,0)
    # X offset
    write_output_float_register(4,0)
    # Z offset
    write_output_float_register(5,0)
    # PLUS Integral
    write_output_float_register(6,0)
    # MINUS Integral
    write_output_float_register(7,0)
    # Standard_Arc_Current
    write_output_float_register(8,0)
    # ALL Integral
    write_output_float_register(9,0)
    # x up
    write_output_float_register(10,0)
    # x ui
    write_output_float_register(11,0)
    # z up
    write_output_float_register(12,0)
    # z ui
    write_output_float_register(13,0)
    # x
    write_output_float_register(14,0)
    # y
    write_output_float_register(15,0)
    # z
    write_output_float_register(16,0)
    # welding on/off polyscope
    write_output_float_register(17,0)
    # touch on/off polyscope
    write_output_float_register(18,0)
    # ratio_t
    write_output_float_register(19,0)
    # get_wcr polyscope
    write_output_float_register(20,0)
    # get_touch polyscope
    write_output_float_register(21,0)
    # write_welder
    write_output_float_register(22,0)
    # MIDDLE_Integral_org
    write_output_float_register(23,0)
    # PLUS Integral_org
    write_output_float_register(24,0)
    # MINUS Integral_org
    write_output_float_register(25,0)

    #init
    global cycle_number = 0
    global cycle_done = False
    global cycle1_plus = 0
    global cycle1_minus = 0
    global cycle1_middle = 0
    global current_to_welding_m = read_port_register(133)
    global voltage_to_welding_m = read_port_register(134)/10
    global c_maxcut = current_to_welding_m*1.2
    global c_mincut = current_to_welding_m*0.8
    global v_maxcut = voltage_to_welding_m*1.2
    global v_mincut = voltage_to_welding_m*0.8
    global Standard_Arc_Current = current_to_welding_m
    global Standard_Arc_voltage = voltage_to_welding_m
    global FB_CURRENT_UR = 0
    global FB_VOLTAGE_UR = 0
    global FB_CURRENT_UR_org = 0
    global FB_VOLTAGE_UR_org = 0
    global one_cycle_p_count = 0
    global one_cycle_m_count = 0
    global one_cycle_p_accum = 0
    global one_cycle_m_accum = 0
    global one_cycle_p_accum_org = 0
    global one_cycle_m_accum_org = 0
    global cal_off_ang_rx = 0
    global cal_off_ang_ry = 0
    global Up = 0
    global Ui = 0
    global Pi_sum = 0
    global Up_z = 0
    global Ui_z = 0
    global Pi_sum_z = 0
    global peak_value = 0
    global ratio_t = 0
    global welding_off_t = 55
    global program_weld_on = False
    global next_path_c = False
    global move_p = [dumy_p,dumy_p,dumy_p]
    global hicomm = True
    global current_on = False
    timer_counter = 0
    sync()
  end

  # get line distance without caring orientation
  def get_line_dist(get_wp1,get_wp2):
    return sqrt((get_wp2[0]-get_wp1[0])*(get_wp2[0]-get_wp1[0])+(get_wp2[1]-get_wp1[1])*(get_wp2[1]-get_wp1[1])+(get_wp2[2]-get_wp1[2])*(get_wp2[2]-get_wp1[2]))
  end

  def plus_minus(num):
    if(num<0):
      return -1
    else:
      return 1
    end
  end

  def get_feature_plane_xz(p1, p2, p3):

    # Step 1. Get the direction vectors
    d12 = [ p2[0]-p1[0], p2[1]-p1[1], p2[2]-p1[2] ]
    d13 = [ p3[0]-p1[0], p3[1]-p1[1], p3[2]-p1[2] ]

    # Step 2. Get the direction vector of Z axis by cross product of d12 and d13
    dy = cross_product(d13, d12)

    # Step 3. Get the X and Z unit direction vectors by normalizing d12 and dz
    temp = norm(d12)
    ux = [ d12[0]/temp, d12[1]/temp, d12[2]/temp ]
    temp = norm(dy)
    uy = [ dy[0]/temp, dy[1]/temp, dy[2]/temp ]

    # Step 4. Get Y unit direction vector by cross product of uz and ux
    uz = cross_product(ux, uy)

    # Step 5. Get the rotation matrix from the unit direction vectors
    rotmat = [ ux[0], ux[1], ux[2], uy[0], uy[1], uy[2], uz[0], uz[1], uz[2] ]

    # Step 6. Get the rotation vector from the rotation matrix
    rotvec = rotmat2rotvec(rotmat)

    # Step 7. Get the feature plane with the origin at p1 and the frame achieved at step 6
    feature_plane = p[ p1[0], p1[1], p1[2], rotvec[0], rotvec[1], rotvec[2] ]

    return feature_plane
  end

  def get_feature_plane_yz(p1, p2, p3):

    # Step 1. Get the direction vectors
    d12 = [ p2[0]-p1[0], p2[1]-p1[1], p2[2]-p1[2] ]
    d13 = [ p3[0]-p1[0], p3[1]-p1[1], p3[2]-p1[2] ]

    # Step 2. Get the direction vector of Z axis by cross product of d12 and d13
    dx = cross_product(d12, d13)

    # Step 3. Get the X and Z unit direction vectors by normalizing d12 and dz
    temp = norm(d12)
    uy = [ d12[0]/temp, d12[1]/temp, d12[2]/temp ]
    temp = norm(dx)
    ux = [ dx[0]/temp, dx[1]/temp, dx[2]/temp ]

    # Step 4. Get Y unit direction vector by cross product of uz and ux
    uz = cross_product(ux, uy)

    # Step 5. Get the rotation matrix from the unit direction vectors
    rotmat = [ ux[0], ux[1], ux[2], uy[0], uy[1], uy[2], uz[0], uz[1], uz[2] ]

    # Step 6. Get the rotation vector from the rotation matrix
    rotvec = rotmat2rotvec(rotmat)

    # Step 7. Get the feature plane with the origin at p1 and the frame achieved at step 6
    feature_plane = p[ p1[0], p1[1], p1[2], rotvec[0], rotvec[1], rotvec[2] ]

    return feature_plane
  end

  def get_feature_plane_xy(p1, p2, p3):

    # Step 1. Get the direction vectors
    d12 = [ p2[0]-p1[0], p2[1]-p1[1], p2[2]-p1[2] ]
    d13 = [ p3[0]-p1[0], p3[1]-p1[1], p3[2]-p1[2] ]

    # Step 2. Get the direction vector of Z axis by cross product of d12 and d13
    dz = cross_product(d12, d13)

    # Step 3. Get the X and Z unit direction vectors by normalizing d12 and dz
    temp = norm(d12)
    ux = [ d12[0]/temp, d12[1]/temp, d12[2]/temp ]
    temp = norm(dz)
    uz = [ dz[0]/temp, dz[1]/temp, dz[2]/temp ]

    # Step 4. Get Y unit direction vector by cross product of uz and ux
    uy = cross_product(uz, ux)

    # Step 5. Get the rotation matrix from the unit direction vectors
    rotmat = [ ux[0], ux[1], ux[2], uy[0], uy[1], uy[2], uz[0], uz[1], uz[2] ]

    # Step 6. Get the rotation vector from the rotation matrix
    rotvec = rotmat2rotvec(rotmat)

    # Step 7. Get the feature plane with the origin at p1 and the frame achieved at step 6
    feature_plane = p[ p1[0], p1[1], p1[2], rotvec[0], rotvec[1], rotvec[2] ]

    return feature_plane
  end

  #### ur_weaving_rev1 by Henry
  #  x_feature = pose_trans(N_Pose,pose_inv(p[0,0,x,0,0,0])
  def feature_offset(fun_pose,fun_offset,fun_plane=p[0,0,0,0,0,0]):
    fun_p_feature = pose_trans ( pose_inv (fun_plane), fun_pose)
    fun_offrot = rotvec2rpy([fun_p_feature[3],fun_p_feature[4],fun_p_feature[5]])
    fun_offset = p[fun_offset[0],fun_offset[1],fun_offset[2],fun_offrot[0]+fun_offset[3],fun_offrot[1]+fun_offset[4],fun_offrot[2]+fun_offset[5]]
    fun_offset_p = p[fun_offset[0],fun_offset[1],fun_offset[2],0,0,0]
    fun_offrpy_rot = rpy2rotvec([fun_offset[3],fun_offset[4],fun_offset[5]])
    fun_offset_rot = p[0,0,0,fun_offrpy_rot[0],fun_offrpy_rot[1],fun_offrpy_rot[2]]
    fun_cal_p = pose_trans(fun_plane,pose_trans(fun_offset_p,fun_p_feature))
    fun_cal_rot = pose_trans(fun_plane,fun_offset_rot)
    result_cal = p[fun_cal_p[0],fun_cal_p[1],fun_cal_p[2],fun_cal_rot[3],fun_cal_rot[4],fun_cal_rot[5]]
    return result_cal
  end

  ## same as changing feature in Move command
  ## Set offset into Plane and move position by it
  def plane_offset(fun_pose,p_offset,fun_plane=p[0,0,0,0,0,0]):
    fun_p_feature = pose_trans ( pose_inv (fun_plane), fun_pose)
    fun_plane = pose_trans(fun_plane,p[p_offset[0],p_offset[1],p_offset[2],0,0,0])
    fun_p_result = pose_trans(pose_trans(fun_plane,p[0,0,0,p_offset[3],p_offset[4],p_offset[5]]),fun_p_feature)
    return fun_p_result
  end

  #  convert from rotation matrix to rotation vector
  ####
  def rotmat2rotvec(rotmat):

    # array to matrix
    r11 = rotmat[0]
    r21 = rotmat[1]
    r31 = rotmat[2]
    r12 = rotmat[3]
    r22 = rotmat[4]
    r32 = rotmat[5]
    r13 = rotmat[6]
    r23 = rotmat[7]
    r33 = rotmat[8]

    # rotation matrix to rotation vector
    theta = acos((r11+r22+r33-1)/2)
    sth = sin(theta)

